C07282=1064.965,385.568,389.284,174.919,35.671,156.670
C07283=1064.957,385.321,389.325,174.915,35.664,156.668
C07284=1064.950,385.075,389.365,174.910,35.657,156.666
C07285=1064.943,384.828,389.405,174.904,35.650,156.665
C07286=1064.936,384.581,389.445,174.899,35.643,156.663
C07287=1064.928,384.334,389.485,174.895,35.636,156.662
C07288=1064.922,384.089,389.526,174.890,35.629,156.660
C07289=1064.914,383.842,389.566,174.884,35.621,156.658
C07290=1064.907,383.595,389.605,174.879,35.615,156.657
C07291=1064.900,383.348,389.646,174.875,35.608,156.655
C07292=1064.893,383.102,389.685,174.870,35.600,156.653
C07293=1064.886,382.855,389.726,174.865,35.594,156.652
C07294=1064.879,382.609,389.765,174.859,35.587,156.650
C07295=1064.871,382.362,389.805,174.855,35.580,156.649
C07296=1064.865,382.115,389.845,174.850,35.573,156.647
C07297=1064.857,381.868,389.885,174.845,35.566,156.645
C07298=1064.850,381.622,389.925,174.840,35.559,156.644
C07299=1064.843,381.376,389.965,174.835,35.552,156.642
C07300=1064.836,381.128,390.004,174.830,35.545,156.641
C07301=1064.829,380.882,390.044,174.825,35.538,156.639
C07302=1064.821,380.635,390.084,174.821,35.532,156.637
C07303=1064.814,380.389,390.123,174.816,35.525,156.636
C07304=1064.807,380.142,390.162,174.810,35.518,156.634
C07305=1064.799,379.895,390.202,174.805,35.511,156.633
C07306=1064.792,379.649,390.242,174.801,35.504,156.631
C07307=1064.785,379.401,390.281,174.796,35.498,156.630
C07308=1064.778,379.155,390.320,174.791,35.491,156.628
C07309=1064.771,378.908,390.359,174.787,35.484,156.627
C07310=1064.763,378.661,390.399,174.781,35.478,156.625
C07311=1064.756,378.415,390.439,174.776,35.471,156.624
C07312=1064.749,378.168,390.478,174.772,35.464,156.622
C07313=1064.742,377.921,390.517,174.767,35.458,156.621
C07314=1064.735,377.675,390.556,174.762,35.451,156.619
C07315=1064.728,377.428,390.595,174.758,35.444,156.617
C07316=1064.721,377.182,390.635,174.753,35.438,156.616
C07317=1064.713,376.934,390.674,174.748,35.432,156.615
C07318=1064.706,376.688,390.713,174.744,35.425,156.613
C07319=1064.700,376.441,390.752,174.738,35.418,156.611
C07320=1064.693,376.194,390.791,174.733,35.411,156.610
C07321=1064.685,375.947,390.831,174.729,35.405,156.609
C07322=1064.678,375.700,390.870,174.724,35.399,156.607
C07323=1064.671,375.454,390.909,174.719,35.392,156.605
C07324=1064.665,375.207,390.948,174.715,35.386,156.604
C07325=1064.657,374.961,390.987,174.710,35.379,156.603
C07326=1064.651,374.714,391.026,174.706,35.372,156.601
C07327=1064.644,374.467,391.065,174.701,35.366,156.600
C07328=1064.636,374.219,391.104,174.696,35.360,156.598
C07329=1064.630,373.973,391.142,174.692,35.353,156.597
C07330=1064.622,373.727,391.181,174.687,35.347,156.595
C07331=1064.616,373.481,391.220,174.683,35.341,156.594
C07332=1064.609,373.235,391.259,174.678,35.334,156.592
C07333=1064.602,372.988,391.298,174.673,35.328,156.591
C07334=1064.595,372.743,391.336,174.669,35.321,156.589
C07335=1064.588,372.496,391.375,174.664,35.315,156.588
C07336=1064.581,372.250,391.414,174.660,35.309,156.587
C07337=1064.574,372.002,391.452,174.655,35.302,156.585
C07338=1064.566,371.756,391.490,174.650,35.296,156.584
C07339=1064.560,371.509,391.529,174.646,35.290,156.582
C07340=1064.553,371.262,391.568,174.641,35.283,156.581
C07341=1064.545,371.016,391.606,174.637,35.277,156.579
C07342=1064.539,370.769,391.645,174.632,35.271,156.578
C07343=1064.532,370.521,391.683,174.627,35.265,156.577
C07344=1064.524,370.275,391.721,174.623,35.259,156.575
C07345=1064.518,370.028,391.760,174.618,35.253,156.574
C07346=1064.511,369.781,391.798,174.614,35.246,156.573
C07347=1064.504,369.534,391.837,174.609,35.240,156.571
C07348=1064.497,369.287,391.875,174.605,35.234,156.570
C07349=1064.490,369.040,391.913,174.600,35.228,156.568
C07350=1064.483,368.793,391.952,174.596,35.222,156.567
C07351=1064.476,368.546,391.990,174.591,35.215,156.566
C07352=1064.469,368.299,392.028,174.586,35.209,156.564
C07353=1064.462,368.052,392.066,174.582,35.204,156.563
C07354=1064.455,367.805,392.105,174.578,35.197,156.562
C07355=1064.449,367.559,392.142,174.574,35.191,156.560
C07356=1064.442,367.312,392.181,174.569,35.185,156.559
C07357=1064.435,367.065,392.219,174.565,35.179,156.557
C07358=1064.428,366.818,392.258,174.560,35.173,156.556
C07359=1064.421,366.571,392.295,174.556,35.167,156.555
C07360=1064.414,366.323,392.333,174.551,35.161,156.553
C07361=1064.407,366.077,392.371,174.547,35.155,156.552
C07362=1064.401,365.830,392.409,174.542,35.149,156.551
C07363=1064.393,365.583,392.447,174.539,35.143,156.549
C07364=1064.387,365.336,392.486,174.534,35.137,156.548
C07365=1064.380,365.089,392.524,174.530,35.131,156.547
C07366=1064.373,364.842,392.561,174.525,35.125,156.545
C07367=1064.367,364.595,392.599,174.521,35.119,156.544
C07368=1064.359,364.348,392.637,174.516,35.113,156.543
C07369=1064.353,364.101,392.675,174.512,35.107,156.541
C07370=1064.346,363.854,392.713,174.508,35.101,156.540
C07371=1064.339,363.607,392.750,174.504,35.095,156.539
C07372=1064.332,363.360,392.788,174.499,35.089,156.537
C07373=1064.325,363.113,392.826,174.495,35.084,156.536
C07374=1064.318,362.866,392.863,174.490,35.078,156.535
C07375=1064.311,362.619,392.900,174.486,35.072,156.533
C07376=1064.305,362.372,392.938,174.482,35.066,156.532
C07377=1064.298,362.125,392.976,174.478,35.060,156.531
C07378=1064.290,361.877,393.013,174.473,35.055,156.530
C07379=1064.284,361.631,393.051,174.469,35.048,156.528
C07380=1064.277,361.384,393.089,174.464,35.043,156.527
C07381=1064.270,361.136,393.126,174.461,35.037,156.526
C07382=1064.264,360.889,393.163,174.456,35.031,156.525
C07383=1064.256,360.642,393.200,174.452,35.026,156.523
C07384=1064.250,360.395,393.238,174.447,35.020,156.522
C07385=1064.243,360.158,393.274,174.444,35.014,156.521
C07386=1064.237,359.920,393.310,174.439,35.009,156.520
C07387=1064.230,359.683,393.346,174.435,35.004,156.518
C07388=1064.224,359.445,393.382,174.431,34.998,156.517
C07389=1064.217,359.208,393.417,174.427,34.992,156.516
C07390=1064.211,358.970,393.453,174.424,34.987,156.515
C07391=1064.204,358.733,393.489,174.419,34.981,156.514
C07392=1064.195,358.386,393.541,174.414,34.974,156.512
C07393=1064.185,358.030,393.595,174.407,34.966,156.510
C07394=1064.178,357.782,393.632,174.403,34.960,156.509
C07395=1064.171,357.535,393.669,174.399,34.954,156.508
C07396=1064.165,357.288,393.706,174.395,34.948,156.506
C07397=1064.157,357.041,393.743,174.390,34.943,156.505
C07398=1064.151,356.793,393.780,174.387,34.938,156.504
C07399=1064.144,356.546,393.817,174.382,34.932,156.503
C07400=1064.137,356.299,393.854,174.378,34.926,156.502
C07401=1064.130,356.052,393.891,174.373,34.921,156.500
C07402=1064.124,355.805,393.928,174.370,34.915,156.499
C07403=1064.117,355.557,393.965,174.366,34.910,156.498
C07404=1064.111,355.310,394.001,174.361,34.904,156.497
C07405=1064.103,355.063,394.039,174.358,34.899,156.496
C07406=1064.097,354.816,394.075,174.353,34.893,156.494
C07407=1064.090,354.568,394.112,174.349,34.887,156.493
C07408=1064.083,354.322,394.149,174.346,34.882,156.492
C07409=1064.076,354.074,394.186,174.341,34.877,156.491
C07410=1064.070,353.827,394.222,174.337,34.871,156.489
C07411=1064.064,353.580,394.259,174.333,34.866,156.488
C07412=1064.056,353.333,394.296,174.329,34.860,156.487
C07413=1064.050,353.086,394.333,174.324,34.855,156.486
C07414=1064.043,352.838,394.369,174.321,34.849,156.485
C07415=1064.037,352.591,394.406,174.317,34.844,156.484
C07416=1064.031,352.344,394.442,174.312,34.838,156.482
C07417=1064.024,352.096,394.479,174.309,34.833,156.481
C07418=1064.017,351.849,394.516,174.304,34.828,156.480
C07419=1064.010,351.602,394.551,174.301,34.822,156.479
C07420=1064.003,351.355,394.588,174.297,34.817,156.478
C07421=1063.997,351.108,394.625,174.292,34.811,156.477
C07422=1063.990,350.860,394.661,174.289,34.806,156.475
C07423=1063.983,350.613,394.697,174.285,34.801,156.474
C07424=1063.977,350.366,394.734,174.280,34.795,156.473
C07425=1063.970,350.118,394.771,174.277,34.790,156.472
C07426=1063.963,349.871,394.807,174.272,34.785,156.471
C07427=1063.956,349.625,394.843,174.269,34.779,156.470
C07428=1063.950,349.377,394.879,174.265,34.774,156.468
C07429=1063.943,349.129,394.915,174.260,34.769,156.467
C07430=1063.936,348.882,394.951,174.257,34.764,156.466
C07431=1063.930,348.635,394.988,174.253,34.759,156.465
C07432=1063.923,348.388,395.025,174.249,34.753,156.464
C07433=1063.917,348.140,395.060,174.245,34.748,156.463
C07434=1063.910,347.893,395.096,174.241,34.743,156.462
C07435=1063.903,347.646,395.133,174.237,34.738,156.461
C07436=1063.897,347.398,395.169,174.233,34.732,156.459
C07437=1063.890,347.151,395.205,174.229,34.727,156.458
C07438=1063.883,346.904,395.241,174.225,34.722,156.457
C07439=1063.877,346.656,395.276,174.222,34.717,156.456
C07440=1063.870,346.409,395.313,174.217,34.712,156.455
C07441=1063.859,345.994,395.373,174.211,34.702,156.453
C07442=1063.848,345.577,395.433,174.204,34.694,156.451
C07443=1063.837,345.161,395.494,174.198,34.685,156.449
C07444=1063.826,344.745,395.554,174.192,34.677,156.448
C07445=1063.819,344.498,395.590,174.188,34.671,156.446
C07446=1063.813,344.250,395.626,174.183,34.666,156.445
C07447=1063.806,344.004,395.662,174.180,34.661,156.444
C07448=1063.800,343.756,395.698,174.176,34.656,156.443
C07449=1063.793,343.508,395.733,174.172,34.651,156.442
C07450=1063.787,343.261,395.769,174.168,34.646,156.441
C07451=1063.780,343.013,395.805,174.165,34.641,156.440
C07452=1063.773,342.766,395.840,174.160,34.636,156.439
C07453=1063.767,342.518,395.876,174.157,34.631,156.438
C07454=1063.760,342.272,395.911,174.154,34.626,156.437
C07455=1063.753,342.024,395.947,174.149,34.621,156.436
C07456=1063.747,341.777,395.982,174.146,34.615,156.434
C07457=1063.740,341.529,396.017,174.142,34.611,156.434
C07458=1063.733,341.282,396.053,174.138,34.606,156.432
C07459=1063.727,341.035,396.089,174.134,34.600,156.431
C07460=1063.720,340.787,396.124,174.131,34.596,156.430
C07461=1063.714,340.540,396.160,174.126,34.591,156.429
C07462=1063.707,340.292,396.195,174.123,34.585,156.428
C07463=1063.701,340.045,396.230,174.119,34.581,156.427
C07464=1063.694,339.798,396.265,174.115,34.575,156.426
C07465=1063.688,339.550,396.301,174.111,34.571,156.425
C07466=1063.681,339.303,396.336,174.108,34.566,156.424
C07467=1063.674,339.055,396.371,174.105,34.560,156.423
C07468=1063.668,338.808,396.407,174.100,34.556,156.422
C07469=1063.662,338.560,396.442,174.097,34.551,156.421
C07470=1063.655,338.313,396.477,174.093,34.546,156.420
C07471=1063.649,338.065,396.513,174.089,34.541,156.419
C07472=1063.642,337.818,396.548,174.086,34.536,156.418
C07473=1063.635,337.570,396.583,174.082,34.531,156.417
C07474=1063.628,337.323,396.618,174.078,34.526,156.416
C07475=1063.622,337.075,396.654,174.074,34.521,156.415
C07476=1063.617,336.828,396.688,174.071,34.516,156.414
C07477=1063.610,336.581,396.723,174.068,34.512,156.413
C07478=1063.603,336.333,396.758,174.063,34.506,156.411
C07479=1063.596,336.086,396.794,174.060,34.502,156.410
C07480=1063.590,335.838,396.828,174.056,34.497,156.409
C07481=1063.583,335.591,396.863,174.052,34.492,156.408
C07482=1063.576,335.343,396.898,174.049,34.487,156.407
C07483=1063.570,335.096,396.933,174.045,34.483,156.406
C07484=1063.563,334.848,396.968,174.042,34.477,156.405
C07485=1063.558,334.601,397.003,174.038,34.473,156.404
C07486=1063.551,334.354,397.038,174.034,34.468,156.403
C07487=1063.544,334.106,397.073,174.031,34.463,156.402
C07488=1063.538,333.858,397.108,174.026,34.458,156.401
C07489=1063.531,333.610,397.142,174.023,34.454,156.400
C07490=1063.525,333.364,397.177,174.020,34.449,156.399
C07491=1063.519,333.116,397.211,174.016,34.444,156.398
C07492=1063.512,332.868,397.247,174.012,34.439,156.397
C07493=1063.505,332.631,397.280,174.009,34.434,156.396
C07494=1063.499,332.393,397.313,174.006,34.430,156.395
C07495=1063.493,332.155,397.347,174.003,34.426,156.395
C07496=1063.487,331.917,397.380,173.998,34.421,156.394
C07497=1063.480,331.680,397.413,173.995,34.416,156.393
C07498=1063.475,331.441,397.446,173.992,34.412,156.392
C07499=1063.468,331.204,397.480,173.989,34.407,156.391
C07500=1063.462,330.966,397.513,173.985,34.402,156.390
C07501=1063.456,330.718,397.547,173.981,34.398,156.389
C07502=1063.449,330.471,397.582,173.978,34.393,156.388
C07503=1063.442,330.223,397.616,173.975,34.388,156.387
C07504=1063.436,329.976,397.650,173.970,34.384,156.386
C07505=1063.429,329.728,397.684,173.967,34.379,156.385
C07506=1063.423,329.481,397.719,173.964,34.375,156.384
C07507=1063.415,329.233,397.753,173.960,34.370,156.383
C07508=1063.410,328.986,397.787,173.956,34.366,156.382
C07509=1063.403,328.738,397.822,173.953,34.361,156.381
C07510=1063.396,328.490,397.856,173.950,34.356,156.380
C07511=1063.389,328.243,397.891,173.946,34.351,156.379
C07512=1063.383,327.995,397.925,173.942,34.347,156.378
C07513=1063.376,327.748,397.959,173.939,34.342,156.377
C07514=1063.370,327.500,397.993,173.935,34.338,156.376
C07515=1063.364,327.252,398.027,173.932,34.333,156.375
C07516=1063.357,327.005,398.061,173.928,34.329,156.374
C07517=1063.350,326.757,398.095,173.925,34.324,156.373
C07518=1063.343,326.510,398.129,173.921,34.319,156.372
C07519=1063.337,326.262,398.163,173.918,34.315,156.371
C07520=1063.331,326.014,398.197,173.914,34.311,156.371
C07521=1063.324,325.767,398.231,173.911,34.306,156.370
C07522=1063.317,325.519,398.266,173.907,34.301,156.369
C07523=1063.311,325.272,398.299,173.904,34.296,156.368
C07524=1063.304,325.024,398.333,173.901,34.292,156.367
C07525=1063.299,324.777,398.367,173.897,34.288,156.366
C07526=1063.291,324.529,398.401,173.893,34.283,156.365
C07527=1063.285,324.281,398.436,173.890,34.278,156.364
C07528=1063.279,324.033,398.468,173.887,34.274,156.363
C07529=1063.272,323.785,398.503,173.883,34.269,156.362
C07530=1063.266,323.538,398.537,173.880,34.265,156.361
C07531=1063.259,323.290,398.571,173.876,34.260,156.360
C07532=1063.253,323.043,398.605,173.873,34.256,156.359
C07533=1063.246,322.795,398.639,173.870,34.251,156.358
C07534=1063.240,322.547,398.672,173.866,34.247,156.357
C07535=1063.233,322.300,398.706,173.863,34.242,156.357
C07536=1063.227,322.053,398.740,173.859,34.238,156.356
C07537=1063.221,321.806,398.773,173.856,34.233,156.355
C07538=1063.215,321.557,398.807,173.852,34.229,156.354
C07539=1063.209,321.310,398.841,173.849,34.224,156.353
C07540=1063.202,321.062,398.875,173.846,34.220,156.352
C07541=1063.196,320.814,398.908,173.843,34.215,156.351
C07542=1063.189,320.566,398.942,173.839,34.211,156.350
C07543=1063.183,320.319,398.975,173.835,34.206,156.349
C07544=1063.177,320.072,399.009,173.832,34.202,156.348
C07545=1063.170,319.824,399.043,173.829,34.197,156.347
C07546=1063.164,319.576,399.076,173.826,34.193,156.346
C07547=1063.157,319.328,399.110,173.823,34.188,156.346
C07548=1063.151,319.080,399.143,173.819,34.184,156.345
C07549=1063.145,318.839,399.176,173.815,34.179,156.344
C07550=1063.139,318.599,399.209,173.812,34.175,156.343
C07551=1063.133,318.358,399.242,173.809,34.171,156.342
C07552=1063.127,318.118,399.274,173.806,34.167,156.341
C07553=1063.121,317.878,399.306,173.802,34.162,156.340
C07554=1063.115,317.637,399.338,173.799,34.158,156.339
C07555=1063.109,317.396,399.371,173.796,34.154,156.338
C07556=1063.103,317.155,399.404,173.793,34.149,156.338
C07557=1063.096,316.908,399.437,173.790,34.145,156.337
C07558=1063.091,316.660,399.470,173.786,34.140,156.336
C07559=1063.084,316.412,399.503,173.783,34.135,156.335
C07560=1063.078,316.164,399.538,173.780,34.131,156.334
C07561=1063.071,315.917,399.570,173.777,34.127,156.333
C07562=1063.066,315.669,399.604,173.774,34.122,156.332
C07563=1063.059,315.421,399.637,173.770,34.118,156.331
C07564=1063.052,315.174,399.670,173.767,34.114,156.330
C07565=1063.047,314.926,399.703,173.763,34.109,156.329
C07566=1063.040,314.679,399.737,173.760,34.105,156.329
C07567=1063.035,314.431,399.770,173.757,34.100,156.328
C07568=1063.028,314.183,399.803,173.753,34.096,156.327
C07569=1063.022,313.935,399.837,173.750,34.091,156.326
C07570=1063.016,313.687,399.869,173.747,34.087,156.325
C07571=1063.010,313.440,399.902,173.744,34.083,156.324
C07572=1063.002,313.192,399.936,173.741,34.079,156.323
C07573=1062.996,312.944,399.969,173.738,34.074,156.322
C07574=1062.990,312.697,400.002,173.734,34.070,156.321
C07575=1062.983,312.449,400.034,173.731,34.066,156.321
C07576=1062.976,312.201,400.067,173.728,34.062,156.320
C07577=1062.970,311.953,400.100,173.725,34.057,156.319
C07578=1062.963,311.706,400.132,173.721,34.053,156.318
C07579=1062.957,311.458,400.165,173.718,34.048,156.317
C07580=1062.951,311.211,400.198,173.714,34.044,156.316
C07581=1062.944,310.962,400.231,173.711,34.040,156.315
C07582=1062.938,310.715,400.264,173.708,34.036,156.315
C07583=1062.932,310.467,400.296,173.705,34.032,156.314
C07584=1062.925,310.219,400.328,173.702,34.027,156.313
C07585=1062.919,309.971,400.361,173.699,34.023,156.312
C07586=1062.912,309.723,400.394,173.695,34.019,156.311
C07587=1062.905,309.476,400.426,173.692,34.015,156.310
C07588=1062.899,309.228,400.459,173.689,34.010,156.310
C07589=1062.893,308.981,400.492,173.686,34.006,156.309
C07590=1062.887,308.732,400.524,173.683,34.002,156.308
C07591=1062.880,308.485,400.557,173.680,33.998,156.307
C07592=1062.874,308.237,400.589,173.676,33.993,156.306
C07593=1062.868,307.990,400.622,173.673,33.989,156.305
C07594=1062.861,307.742,400.655,173.670,33.985,156.304
C07595=1062.855,307.494,400.686,173.667,33.981,156.304
C07596=1062.848,307.247,400.719,173.664,33.977,156.303
C07597=1062.842,306.999,400.752,173.661,33.972,156.302
C07598=1062.835,306.750,400.784,173.657,33.968,156.301
C07599=1062.829,306.502,400.817,173.654,33.964,156.300
C07600=1062.823,306.255,400.850,173.651,33.960,156.299
C07601=1062.816,306.007,400.881,173.648,33.955,156.298
C07602=1062.810,305.759,400.914,173.645,33.951,156.298
C07603=1062.804,305.512,400.947,173.642,33.947,156.297
C07604=1062.798,305.264,400.978,173.638,33.943,156.296
C07605=1062.791,305.025,401.010,173.635,33.939,156.295
C07606=1062.785,304.786,401.041,173.632,33.935,156.294
C07607=1062.779,304.547,401.072,173.629,33.931,156.294
C07608=1062.774,304.308,401.103,173.626,33.927,156.293
C07609=1062.767,304.070,401.135,173.623,33.922,156.292
C07610=1062.761,303.831,401.166,173.620,33.918,156.291
C07611=1062.755,303.592,401.196,173.618,33.915,156.290
C07612=1062.750,303.354,401.227,173.614,33.911,156.290
C07613=1062.743,303.106,401.259,173.611,33.906,156.289
C07614=1062.737,302.858,401.291,173.608,33.902,156.288
C07615=1062.731,302.611,401.324,173.605,33.898,156.287
C07616=1062.725,302.362,401.356,173.602,33.894,156.286
C07617=1062.719,302.115,401.389,173.599,33.889,156.285
C07618=1062.712,301.867,401.420,173.595,33.885,156.284
C07619=1062.706,301.619,401.452,173.592,33.881,156.284
C07620=1062.700,301.372,401.485,173.589,33.877,156.283
C07621=1062.694,301.123,401.517,173.586,33.872,156.282
C07622=1062.688,300.876,401.548,173.583,33.868,156.281
C07623=1062.681,300.628,401.581,173.581,33.864,156.280
C07624=1062.675,300.380,401.613,173.578,33.860,156.279
C07625=1062.669,300.132,401.645,173.575,33.856,156.279
C07626=1062.663,299.885,401.677,173.571,33.852,156.278
C07627=1062.657,299.637,401.709,173.568,33.847,156.277
C07628=1062.651,299.389,401.741,173.565,33.843,156.276
C07629=1062.645,299.140,401.773,173.562,33.839,156.275
C07630=1062.638,298.892,401.804,173.559,33.835,156.274
C07631=1062.632,298.646,401.837,173.556,33.831,156.274
C07632=1062.626,298.397,401.869,173.553,33.826,156.273
C07633=1062.620,298.149,401.901,173.550,33.822,156.272
C07634=1062.614,297.902,401.932,173.547,33.818,156.271
C07635=1062.608,297.654,401.964,173.544,33.814,156.270
C07636=1062.602,297.405,401.996,173.541,33.810,156.270
C07637=1062.595,297.158,402.028,173.538,33.806,156.269
C07638=1062.590,296.911,402.060,173.535,33.801,156.268
C07639=1062.583,296.663,402.091,173.532,33.797,156.267
C07640=1062.577,296.415,402.123,173.530,33.793,156.266
C07641=1062.571,296.167,402.155,173.526,33.790,156.265
C07642=1062.565,295.918,402.187,173.523,33.785,156.265
C07643=1062.558,295.671,402.218,173.520,33.781,156.264
C07644=1062.552,295.423,402.250,173.517,33.777,156.263
C07645=1062.546,295.175,402.281,173.514,33.773,156.262
C07646=1062.541,294.927,402.312,173.511,33.769,156.261
C07647=1062.534,294.679,402.344,173.508,33.765,156.261
C07648=1062.527,294.431,402.375,173.506,33.761,156.260
C07649=1062.521,294.183,402.407,173.502,33.757,156.259
C07650=1062.515,293.936,402.438,173.499,33.752,156.258
C07651=1062.508,293.688,402.470,173.496,33.749,156.257
C07652=1062.502,293.440,402.502,173.493,33.745,156.257
C07653=1062.496,293.191,402.532,173.490,33.740,156.256
C07654=1062.490,292.944,402.563,173.488,33.736,156.255
C07655=1062.484,292.696,402.595,173.485,33.733,156.254
C07656=1062.477,292.448,402.627,173.482,33.728,156.253
C07657=1062.471,292.201,402.658,173.479,33.724,156.253
C07658=1062.465,291.952,402.689,173.475,33.720,156.252
C07659=1062.459,291.704,402.721,173.472,33.716,156.251
C07660=1062.452,291.457,402.752,173.470,33.712,156.250
C07661=1062.447,291.225,402.780,173.467,33.709,156.250
C07662=1062.440,290.994,402.810,173.464,33.704,156.249
C07663=1062.435,290.763,402.838,173.462,33.701,156.248
C07664=1062.429,290.532,402.868,173.459,33.697,156.247
C07665=1062.423,290.300,402.897,173.456,33.694,156.247
C07666=1062.417,290.069,402.926,173.454,33.689,156.246
C07667=1062.412,289.838,402.955,173.450,33.686,156.245
C07668=1062.406,289.607,402.984,173.448,33.682,156.244
C07669=1062.400,289.359,403.015,173.445,33.678,156.244
C07670=1062.394,289.111,403.047,173.442,33.674,156.243
C07671=1062.388,288.862,403.077,173.439,33.670,156.242
C07672=1062.381,288.615,403.109,173.437,33.666,156.241
C07673=1062.375,288.366,403.139,173.434,33.662,156.240
C07674=1062.369,288.119,403.170,173.431,33.658,156.240
C07675=1062.362,287.871,403.201,173.428,33.654,156.239
C07676=1062.356,287.623,403.232,173.425,33.650,156.238
C07677=1062.350,287.375,403.263,173.422,33.646,156.237
C07678=1062.343,287.127,403.294,173.419,33.642,156.237
C07679=1062.337,286.879,403.325,173.416,33.638,156.236
C07680=1062.331,286.631,403.355,173.413,33.634,156.235
C07681=1062.324,286.383,403.387,173.411,33.630,156.234
C07682=1062.318,286.135,403.417,173.408,33.626,156.233
C07683=1062.312,285.887,403.449,173.405,33.622,156.233
C07684=1062.306,285.639,403.479,173.402,33.618,156.232
C07685=1062.300,285.390,403.510,173.399,33.614,156.231
C07686=1062.294,285.143,403.541,173.397,33.610,156.230
C07687=1062.288,284.895,403.572,173.394,33.606,156.230
C07688=1062.282,284.647,403.602,173.390,33.602,156.229
C07689=1062.275,284.398,403.633,173.388,33.599,156.228
C07690=1062.269,284.152,403.663,173.385,33.594,156.227
C07691=1062.262,283.903,403.694,173.382,33.590,156.226
C07692=1062.256,283.655,403.725,173.379,33.586,156.226
C07693=1062.250,283.407,403.755,173.377,33.582,156.225
C07694=1062.244,283.159,403.786,173.374,33.579,156.224
C07695=1062.237,282.911,403.817,173.371,33.574,156.223
C07696=1062.232,282.663,403.847,173.368,33.570,156.223
C07697=1062.225,282.415,403.878,173.366,33.567,156.222
C07698=1062.219,282.167,403.908,173.363,33.562,156.221
C07699=1062.213,281.919,403.939,173.359,33.559,156.220
C07700=1062.207,281.670,403.970,173.357,33.555,156.220
C07701=1062.201,281.423,404.000,173.354,33.550,156.219
C07702=1062.195,281.175,404.031,173.351,33.547,156.218
C07703=1062.189,280.927,404.062,173.349,33.543,156.217
C07704=1062.183,280.679,404.092,173.346,33.539,156.217
C07705=1062.176,280.431,404.123,173.343,33.535,156.216
C07706=1062.171,280.183,404.153,173.340,33.530,156.215
C07707=1062.164,279.934,404.184,173.338,33.527,156.214
C07708=1062.158,279.687,404.214,173.335,33.523,156.213
C07709=1062.152,279.439,404.244,173.332,33.519,156.213
C07710=1062.145,279.190,404.275,173.330,33.515,156.212
C07711=1062.140,278.942,404.304,173.326,33.511,156.211
C07712=1062.133,278.694,404.334,173.323,33.507,156.210
C07713=1062.127,278.446,404.365,173.321,33.503,156.210
C07714=1062.121,278.198,404.395,173.318,33.499,156.209
C07715=1062.115,277.950,404.426,173.315,33.495,156.208
C07716=1062.108,277.702,404.456,173.313,33.491,156.207
C07717=1062.103,277.476,404.484,173.310,33.488,156.207
C07718=1062.097,277.250,404.511,173.308,33.485,156.206
C07719=1062.091,277.024,404.538,173.305,33.481,156.205
C07720=1062.085,276.799,404.566,173.303,33.477,156.205
C07721=1062.081,276.572,404.593,173.301,33.474,156.204
C07722=1062.075,276.347,404.620,173.298,33.470,156.203
C07723=1062.070,276.121,404.648,173.296,33.466,156.203
C07724=1062.063,275.895,404.675,173.293,33.463,156.202
C07725=1062.057,275.647,404.706,173.291,33.459,156.201
C07726=1062.052,275.398,404.735,173.287,33.455,156.200
C07727=1062.045,275.150,404.765,173.284,33.451,156.200
C07728=1062.039,274.902,404.796,173.282,33.447,156.199
C07729=1062.033,274.655,404.826,173.279,33.443,156.198
C07730=1062.027,274.406,404.855,173.276,33.439,156.197
C07731=1062.020,274.158,404.886,173.274,33.436,156.197
C07732=1062.014,273.910,404.915,173.271,33.431,156.196
C07733=1062.008,273.662,404.945,173.269,33.428,156.195
C07734=1062.002,273.413,404.976,173.266,33.424,156.194
C07735=1061.995,273.165,405.005,173.263,33.420,156.194
C07736=1061.990,272.917,405.035,173.261,33.416,156.193
C07737=1061.983,272.669,405.064,173.258,33.412,156.192
C07738=1061.977,272.421,405.095,173.256,33.408,156.191
C07739=1061.970,272.173,405.125,173.253,33.404,156.191
C07740=1061.965,271.925,405.155,173.250,33.400,156.190
C07741=1061.958,271.677,405.184,173.247,33.396,156.189
C07742=1061.952,271.428,405.214,173.244,33.393,156.188
C07743=1061.946,271.180,405.243,173.242,33.388,156.188
C07744=1061.940,270.932,405.274,173.239,33.385,156.187
C07745=1061.934,270.684,405.303,173.236,33.381,156.186
C07746=1061.928,270.436,405.333,173.234,33.377,156.185
C07747=1061.921,270.187,405.362,173.231,33.373,156.185
C07748=1061.915,269.940,405.393,173.229,33.369,156.184
C07749=1061.909,269.691,405.422,173.226,33.365,156.183
C07750=1061.904,269.443,405.451,173.223,33.361,156.182
C07751=1061.897,269.196,405.481,173.221,33.357,156.182
C07752=1061.891,268.947,405.510,173.218,33.354,156.181
C07753=1061.885,268.698,405.540,173.216,33.350,156.180
C07754=1061.878,268.451,405.570,173.213,33.346,156.179
C07755=1061.873,268.202,405.600,173.211,33.342,156.179
C07756=1061.866,267.954,405.629,173.208,33.338,156.178
C07757=1061.860,267.707,405.658,173.205,33.334,156.177
C07758=1061.854,267.458,405.688,173.203,33.330,156.176
C07759=1061.848,267.209,405.718,173.199,33.327,156.176
C07760=1061.841,266.961,405.747,173.197,33.323,156.175
C07761=1061.835,266.714,405.776,173.194,33.319,156.174
C07762=1061.829,266.465,405.806,173.192,33.315,156.173
C07763=1061.823,266.217,405.835,173.189,33.311,156.173
C07764=1061.817,265.969,405.864,173.187,33.307,156.172
C07765=1061.811,265.721,405.894,173.184,33.303,156.171
C07766=1061.805,265.472,405.923,173.181,33.299,156.170
C07767=1061.798,265.224,405.953,173.179,33.296,156.170
C07768=1061.792,264.976,405.982,173.176,33.291,156.169
C07769=1061.786,264.728,406.012,173.174,33.288,156.168
C07770=1061.780,264.480,406.041,173.171,33.284,156.168
C07771=1061.774,264.231,406.070,173.169,33.280,156.167
C07772=1061.768,263.983,406.099,173.166,33.276,156.166
C07773=1061.763,263.759,406.125,173.164,33.273,156.165
C07774=1061.756,263.535,406.152,173.162,33.269,156.165
C07775=1061.752,263.311,406.178,173.159,33.265,156.164
C07776=1061.746,263.087,406.205,173.157,33.262,156.163
C07777=1061.740,262.863,406.231,173.155,33.259,156.163
C07778=1061.734,262.639,406.257,173.153,33.256,156.162
C07779=1061.728,262.415,406.283,173.150,33.252,156.161
C07780=1061.722,262.191,406.309,173.148,33.248,156.161
C07781=1061.716,261.943,406.338,173.146,33.245,156.160
C07782=1061.710,261.694,406.367,173.143,33.241,156.159
C07783=1061.704,261.446,406.396,173.139,33.237,156.159
C07784=1061.698,261.198,406.425,173.137,33.233,156.158
C07785=1061.691,260.950,406.454,173.134,33.229,156.157
C07786=1061.685,260.702,406.483,173.132,33.226,156.156
C07787=1061.679,260.453,406.512,173.129,33.222,156.156
C07788=1061.673,260.205,406.541,173.127,33.218,156.155
C07789=1061.667,259.957,406.569,173.124,33.214,156.154
C07790=1061.660,259.708,406.598,173.122,33.210,156.154
C07791=1061.653,259.461,406.627,173.119,33.207,156.153
C07792=1061.647,259.212,406.656,173.117,33.203,156.152
C07793=1061.641,258.964,406.685,173.114,33.199,156.151
C07794=1061.635,258.716,406.713,173.112,33.195,156.151
C07795=1061.629,258.467,406.742,173.110,33.191,156.150
C07796=1061.622,258.219,406.771,173.107,33.187,156.149
C07797=1061.617,257.971,406.800,173.105,33.184,156.149
C07798=1061.610,257.722,406.829,173.102,33.180,156.148
C07799=1061.604,257.474,406.858,173.100,33.176,156.147
C07800=1061.598,257.226,406.886,173.097,33.172,156.146
C07801=1061.592,256.977,406.915,173.095,33.168,156.146
C07802=1061.585,256.730,406.944,173.092,33.164,156.145
C07803=1061.579,256.481,406.972,173.090,33.161,156.144
C07804=1061.573,256.233,407.001,173.087,33.157,156.143
C07805=1061.566,255.985,407.030,173.085,33.153,156.143
C07806=1061.560,255.736,407.058,173.082,33.149,156.142
C07807=1061.554,255.488,407.087,173.080,33.145,156.141
C07808=1061.549,255.240,407.115,173.078,33.141,156.140
C07809=1061.543,254.991,407.144,173.075,33.137,156.140
C07810=1061.536,254.743,407.172,173.073,33.134,156.139
C07811=1061.530,254.495,407.201,173.070,33.130,156.138
C07812=1061.523,254.247,407.230,173.068,33.126,156.138
C07813=1061.517,253.998,407.258,173.065,33.122,156.137
C07814=1061.511,253.750,407.287,173.063,33.118,156.136
C07815=1061.505,253.501,407.316,173.061,33.114,156.135
C07816=1061.500,253.253,407.344,173.058,33.111,156.135
C07817=1061.493,253.005,407.372,173.056,33.106,156.134
C07818=1061.487,252.757,407.401,173.053,33.103,156.133
C07819=1061.481,252.508,407.430,173.050,33.099,156.133
C07820=1061.475,252.260,407.458,173.048,33.095,156.132
C07821=1061.469,252.012,407.487,173.045,33.091,156.131
C07822=1061.463,251.763,407.515,173.043,33.087,156.130
C07823=1061.457,251.515,407.543,173.040,33.083,156.130
C07824=1061.450,251.267,407.572,173.038,33.079,156.129
C07825=1061.444,251.018,407.600,173.036,33.076,156.128
C07826=1061.438,250.769,407.628,173.033,33.072,156.127
C07827=1061.433,250.522,407.657,173.031,33.068,156.127
C07828=1061.426,250.274,407.685,173.028,33.064,156.126
C07829=1061.421,250.048,407.711,173.026,33.061,156.125
C07830=1061.415,249.823,407.737,173.024,33.057,156.125
C07831=1061.409,249.598,407.762,173.022,33.053,156.124
C07832=1061.405,249.372,407.788,173.020,33.050,156.123
C07833=1061.399,249.148,407.813,173.018,33.046,156.123
C07834=1061.394,248.923,407.839,173.016,33.043,156.122
C07835=1061.389,248.698,407.865,173.013,33.039,156.121
C07836=1061.383,248.473,407.891,173.011,33.036,156.121
C07837=1061.377,248.224,407.919,173.009,33.031,156.120
C07838=1061.371,247.977,407.946,173.007,33.028,156.119
C07839=1061.365,247.728,407.975,173.004,33.024,156.118
C07840=1061.359,247.479,408.003,173.002,33.020,156.118
C07841=1061.353,247.231,408.031,172.999,33.016,156.117
C07842=1061.346,246.983,408.060,172.997,33.012,156.116
C07843=1061.341,246.734,408.088,172.995,33.008,156.115
C07844=1061.335,246.486,408.116,172.992,33.004,156.115
C07845=1061.329,246.238,408.144,172.990,33.000,156.114
C07846=1061.323,245.989,408.172,172.988,32.997,156.113
C07847=1061.317,245.740,408.200,172.985,32.992,156.112
C07848=1061.311,245.493,408.228,172.983,32.989,156.112
C07849=1061.305,245.244,408.256,172.981,32.985,156.111
C07850=1061.298,244.996,408.284,172.978,32.981,156.110
C07851=1061.293,244.747,408.312,172.976,32.977,156.110
C07852=1061.286,244.499,408.339,172.974,32.973,156.109
C07853=1061.280,244.250,408.368,172.971,32.969,156.108
C07854=1061.275,244.002,408.396,172.969,32.965,156.107
C07855=1061.268,243.754,408.423,172.967,32.962,156.107
C07856=1061.262,243.505,408.452,172.964,32.957,156.106
C07857=1061.256,243.257,408.479,172.962,32.954,156.105
C07858=1061.250,243.009,408.507,172.960,32.950,156.104
C07859=1061.243,242.760,408.535,172.958,32.946,156.104
C07860=1061.238,242.512,408.563,172.955,32.942,156.103
C07861=1061.231,242.264,408.591,172.953,32.938,156.102
C07862=1061.226,242.016,408.619,172.951,32.934,156.102
C07863=1061.220,241.767,408.646,172.948,32.931,156.101
C07864=1061.213,241.518,408.673,172.946,32.926,156.100
C07865=1061.207,241.269,408.702,172.944,32.923,156.099
C07866=1061.201,241.022,408.729,172.941,32.919,156.099
C07867=1061.194,240.773,408.757,172.939,32.915,156.098
C07868=1061.189,240.524,408.784,172.937,32.911,156.097
C07869=1061.182,240.276,408.812,172.934,32.907,156.096
C07870=1061.176,240.028,408.840,172.932,32.904,156.096
C07871=1061.170,239.780,408.867,172.930,32.899,156.095
C07872=1061.164,239.530,408.895,172.928,32.896,156.094
C07873=1061.158,239.283,408.922,172.925,32.892,156.094
C07874=1061.151,239.034,408.950,172.923,32.888,156.093
C07875=1061.146,238.785,408.977,172.921,32.884,156.092
C07876=1061.140,238.537,409.005,172.918,32.880,156.091
C07877=1061.133,238.289,409.032,172.916,32.876,156.091
C07878=1061.127,238.040,409.059,172.914,32.873,156.090
C07879=1061.121,237.792,409.087,172.912,32.869,156.089
C07880=1061.115,237.544,409.115,172.909,32.865,156.088
C07881=1061.109,237.295,409.142,172.907,32.861,156.088
C07882=1061.102,237.046,409.169,172.905,32.857,156.087
C07883=1061.096,236.799,409.197,172.903,32.853,156.086
C07884=1061.090,236.549,409.224,172.900,32.849,156.086
C07885=1061.084,236.322,409.249,172.898,32.846,156.085
C07886=1061.079,236.093,409.274,172.896,32.842,156.084
C07887=1061.073,235.865,409.300,172.894,32.839,156.084
C07888=1061.068,235.637,409.324,172.892,32.835,156.083
C07889=1061.063,235.409,409.350,172.890,32.832,156.082
C07890=1061.057,235.181,409.375,172.888,32.828,156.082
C07891=1061.052,234.953,409.400,172.886,32.824,156.081
C07892=1061.045,234.725,409.425,172.884,32.821,156.080
C07893=1061.040,234.476,409.453,172.882,32.817,156.080
C07894=1061.034,234.227,409.479,172.879,32.813,156.079
C07895=1061.027,233.979,409.507,172.877,32.809,156.078
C07896=1061.021,233.731,409.534,172.875,32.805,156.077
C07897=1061.015,233.482,409.562,172.873,32.801,156.077
C07898=1061.009,233.234,409.588,172.871,32.797,156.076
C07899=1061.004,232.985,409.615,172.869,32.794,156.075
C07900=1060.997,232.737,409.643,172.867,32.789,156.074
C07901=1060.991,232.488,409.670,172.865,32.786,156.074
C07902=1060.985,232.239,409.697,172.863,32.781,156.073
C07903=1060.979,231.992,409.724,172.860,32.778,156.072
C07904=1060.973,231.742,409.751,172.858,32.774,156.072
C07905=1060.966,231.495,409.779,172.856,32.770,156.071
C07906=1060.960,231.246,409.806,172.854,32.766,156.070
C07907=1060.954,230.997,409.832,172.851,32.762,156.069
C07908=1060.948,230.749,409.859,172.849,32.758,156.069
C07909=1060.942,230.501,409.887,172.847,32.754,156.068
C07910=1060.936,230.252,409.913,172.845,32.750,156.067
C07911=1060.930,230.003,409.940,172.843,32.747,156.066
C07912=1060.924,229.755,409.967,172.840,32.743,156.066
C07913=1060.918,229.507,409.994,172.838,32.739,156.065
C07914=1060.911,229.258,410.021,172.836,32.735,156.064
C07915=1060.906,229.010,410.048,172.834,32.731,156.063
C07916=1060.899,228.761,410.075,172.832,32.727,156.063
C07917=1060.894,228.512,410.102,172.830,32.723,156.062
C07918=1060.886,228.264,410.129,172.827,32.720,156.061
C07919=1060.880,228.016,410.155,172.825,32.715,156.061
C07920=1060.875,227.767,410.182,172.823,32.712,156.060
C07921=1060.868,227.518,410.209,172.821,32.707,156.059
C07922=1060.862,227.270,410.236,172.819,32.704,156.058
C07923=1060.857,227.022,410.262,172.816,32.700,156.058
C07924=1060.850,226.773,410.289,172.814,32.696,156.057
C07925=1060.844,226.524,410.315,172.812,32.692,156.056
C07926=1060.837,226.275,410.342,172.810,32.688,156.056
C07927=1060.832,226.027,410.369,172.808,32.684,156.055
C07928=1060.826,225.779,410.396,172.806,32.680,156.054
C07929=1060.819,225.530,410.423,172.803,32.676,156.053
C07930=1060.813,225.282,410.449,172.801,32.672,156.053
C07931=1060.807,225.033,410.476,172.799,32.669,156.052
C07932=1060.801,224.784,410.503,172.798,32.664,156.051
C07933=1060.795,224.536,410.529,172.796,32.661,156.050
C07934=1060.789,224.287,410.556,172.794,32.657,156.050
C07935=1060.783,224.039,410.582,172.792,32.653,156.049
C07936=1060.776,223.790,410.609,172.789,32.649,156.048
C07937=1060.771,223.542,410.636,172.787,32.645,156.048
C07938=1060.765,223.294,410.662,172.785,32.641,156.047
C07939=1060.758,223.045,410.689,172.783,32.637,156.046
C07940=1060.752,222.796,410.715,172.781,32.633,156.045
C07941=1060.747,222.565,410.740,172.779,32.630,156.045
C07942=1060.741,222.333,410.765,172.777,32.626,156.044
C07943=1060.735,222.100,410.790,172.775,32.622,156.043
C07944=1060.730,221.868,410.814,172.773,32.618,156.043
C07945=1060.724,221.636,410.839,172.771,32.615,156.042
C07946=1060.718,221.404,410.864,172.769,32.611,156.041
C07947=1060.713,221.172,410.889,172.767,32.607,156.040
C07948=1060.707,220.939,410.913,172.765,32.603,156.040
C07949=1060.701,220.691,410.939,172.763,32.600,156.039
C07950=1060.694,220.442,410.966,172.761,32.596,156.038
C07951=1060.688,220.194,410.992,172.759,32.592,156.038
C07952=1060.682,219.945,411.018,172.757,32.588,156.037
C07953=1060.677,219.697,411.045,172.754,32.584,156.036
C07954=1060.670,219.448,411.071,172.752,32.580,156.035
C07955=1060.664,219.199,411.097,172.750,32.576,156.035
C07956=1060.658,218.951,411.123,172.749,32.572,156.034
C07957=1060.652,218.703,411.150,172.747,32.568,156.033
C07958=1060.645,218.454,411.176,172.745,32.565,156.033
C07959=1060.639,218.205,411.202,172.743,32.560,156.032
C07960=1060.633,217.957,411.228,172.741,32.557,156.031
C07961=1060.627,217.709,411.255,172.739,32.552,156.030
C07962=1060.621,217.460,411.280,172.737,32.549,156.030
C07963=1060.614,217.211,411.307,172.734,32.544,156.029
C07964=1060.608,216.962,411.333,172.732,32.541,156.028
C07965=1060.602,216.714,411.359,172.730,32.536,156.027
C07966=1060.596,216.466,411.385,172.728,32.533,156.027
C07967=1060.590,216.217,411.411,172.726,32.528,156.026
C07968=1060.584,215.969,411.437,172.724,32.525,156.025
C07969=1060.578,215.720,411.463,172.722,32.520,156.024
C07970=1060.571,215.471,411.490,172.720,32.517,156.024
C07971=1060.566,215.222,411.516,172.718,32.512,156.023
C07972=1060.559,214.974,411.542,172.716,32.509,156.022
C07973=1060.554,214.725,411.568,172.714,32.505,156.021
C07974=1060.547,214.477,411.594,172.712,32.501,156.021
C07975=1060.542,214.228,411.620,172.711,32.497,156.020
C07976=1060.535,213.980,411.646,172.709,32.493,156.019
C07977=1060.530,213.731,411.671,172.707,32.489,156.019
C07978=1060.523,213.483,411.698,172.704,32.485,156.018
C07979=1060.518,213.234,411.723,172.702,32.481,156.017
C07980=1060.511,212.985,411.750,172.700,32.477,156.016
C07981=1060.505,212.737,411.775,172.698,32.473,156.016
C07982=1060.499,212.488,411.802,172.696,32.469,156.015
C07983=1060.493,212.240,411.827,172.694,32.465,156.014
C07984=1060.486,211.991,411.853,172.692,32.461,156.013
C07985=1060.481,211.743,411.879,172.690,32.457,156.013
C07986=1060.474,211.494,411.905,172.688,32.453,156.012
C07987=1060.468,211.245,411.930,172.686,32.449,156.011
C07988=1060.462,210.997,411.957,172.684,32.445,156.010
C07989=1060.456,210.748,411.982,172.682,32.441,156.010
C07990=1060.450,210.500,412.007,172.681,32.437,156.009
C07991=1060.444,210.251,412.034,172.679,32.433,156.008
C07992=1060.438,210.002,412.059,172.677,32.428,156.007
C07993=1060.432,209.754,412.085,172.675,32.425,156.007
C07994=1060.426,209.505,412.110,172.673,32.420,156.006
C07995=1060.420,209.257,412.137,172.671,32.417,156.005
C07996=1060.414,209.008,412.162,172.669,32.413,156.004
C07997=1060.408,208.778,412.185,172.667,32.409,156.004
C07998=1060.403,208.549,412.209,172.665,32.405,156.003
C07999=1060.396,208.319,412.233,172.663,32.401,156.002
C08000=1060.391,208.090,412.256,172.661,32.398,156.002
C08001=1060.385,207.860,412.280,172.660,32.394,156.001
C08002=1060.380,207.630,412.303,172.658,32.390,156.000
C08003=1060.373,207.401,412.327,172.656,32.387,156.000
C08004=1060.368,207.170,412.351,172.654,32.383,155.999
C08005=1060.344,206.122,412.455,172.475,32.298,155.990
C08006=1060.337,205.873,412.480,172.472,32.295,155.989
C08007=1060.331,205.625,412.504,172.470,32.292,155.989
C08008=1060.325,205.375,412.529,172.468,32.289,155.988
C08009=1060.319,205.127,412.554,172.465,32.286,155.988
C08010=1060.314,204.878,412.578,172.463,32.282,155.987
C08011=1060.308,204.629,412.604,172.460,32.279,155.987
C08012=1060.302,204.381,412.628,172.458,32.276,155.986
C08013=1060.296,204.132,412.652,172.456,32.273,155.985
C08014=1060.290,203.884,412.677,172.453,32.270,155.985
C08015=1060.284,203.635,412.701,172.451,32.267,155.984
C08016=1060.279,203.386,412.726,172.449,32.263,155.984
C08017=1060.273,203.137,412.750,172.447,32.261,155.983
C08018=1060.267,202.889,412.775,172.445,32.258,155.983
C08019=1060.262,202.639,412.800,172.443,32.254,155.982
C08020=1060.256,202.391,412.824,172.440,32.251,155.982
C08021=1060.249,202.142,412.849,172.438,32.248,155.981
C08022=1060.243,201.893,412.874,172.436,32.245,155.981
C08023=1060.238,201.645,412.898,172.433,32.242,155.980
C08024=1060.231,201.396,412.922,172.431,32.239,155.980
C08025=1060.226,201.147,412.946,172.428,32.236,155.979
C08026=1060.220,200.898,412.970,172.426,32.233,155.979
C08027=1060.214,200.650,412.995,172.424,32.230,155.978
C08028=1060.207,200.401,413.019,172.422,32.227,155.978
C08029=1060.202,200.153,413.043,172.420,32.224,155.977
C08030=1060.195,199.904,413.067,172.418,32.220,155.977
C08031=1060.190,199.655,413.092,172.415,32.218,155.976
C08032=1060.184,199.406,413.116,172.413,32.215,155.976
C08033=1060.178,199.157,413.140,172.411,32.211,155.975
C08034=1060.172,198.908,413.165,172.408,32.209,155.975
C08035=1060.166,198.660,413.188,172.406,32.205,155.974
C08036=1060.160,198.411,413.213,172.404,32.202,155.974
C08037=1060.154,198.162,413.236,172.401,32.199,155.973
C08038=1060.148,197.913,413.261,172.399,32.196,155.973
C08039=1060.142,197.665,413.285,172.397,32.193,155.972
C08040=1060.136,197.415,413.309,172.395,32.190,155.971
C08041=1060.130,197.167,413.333,172.393,32.187,155.971
C08042=1060.124,196.918,413.358,172.391,32.184,155.970
C08043=1060.118,196.670,413.381,172.388,32.181,155.970
C08044=1060.113,196.420,413.406,172.386,32.178,155.970
C08045=1060.106,196.172,413.430,172.384,32.175,155.969
C08046=1060.101,195.923,413.454,172.382,32.172,155.968
C08047=1060.095,195.674,413.478,172.379,32.169,155.968
C08048=1060.089,195.426,413.502,172.377,32.166,155.967
C08049=1060.083,195.177,413.526,172.375,32.163,155.967
C08050=1060.077,194.928,413.550,172.373,32.160,155.967
C08051=1060.071,194.680,413.574,172.371,32.157,155.966
C08052=1060.066,194.430,413.598,172.369,32.154,155.965
C08053=1060.060,194.182,413.622,172.366,32.151,155.965
C08054=1060.054,193.933,413.646,172.364,32.148,155.964
C08055=1060.048,193.684,413.670,172.362,32.145,155.964
C08056=1060.042,193.436,413.694,172.360,32.142,155.963
C08057=1060.036,193.187,413.718,172.357,32.139,155.963
C08058=1060.031,192.937,413.742,172.355,32.136,155.962
C08059=1060.025,192.689,413.765,172.353,32.133,155.962
C08060=1060.019,192.440,413.790,172.351,32.130,155.961
C08061=1060.013,192.192,413.814,172.349,32.127,155.961
C08062=1060.007,191.943,413.837,172.347,32.124,155.960
C08063=1060.002,191.694,413.861,172.345,32.121,155.960
C08064=1059.995,191.445,413.885,172.343,32.118,155.959
C08065=1059.990,191.197,413.909,172.340,32.115,155.959
C08066=1059.982,190.878,413.940,172.337,32.111,155.958
C08067=1059.975,190.558,413.971,172.335,32.108,155.958
C08068=1059.967,190.240,414.001,172.332,32.104,155.957
C08069=1059.960,189.920,414.030,172.329,32.100,155.956
C08070=1059.955,189.671,414.055,172.328,32.097,155.956
C08071=1059.948,189.423,414.079,172.325,32.094,155.955
C08072=1059.943,189.173,414.102,172.323,32.091,155.955
C08073=1059.937,188.925,414.126,172.321,32.088,155.954
C08074=1059.932,188.676,414.150,172.319,32.085,155.954
C08075=1059.925,188.427,414.174,172.316,32.082,155.953
C08076=1059.919,188.179,414.197,172.314,32.079,155.953
C08077=1059.914,187.930,414.221,172.312,32.076,155.952
C08078=1059.908,187.681,414.244,172.310,32.073,155.952
C08079=1059.903,187.432,414.269,172.307,32.070,155.951
C08080=1059.897,187.183,414.292,172.306,32.067,155.951
C08081=1059.891,186.935,414.316,172.304,32.064,155.950
C08082=1059.886,186.685,414.339,172.302,32.061,155.950
C08083=1059.879,186.437,414.363,172.300,32.058,155.949
C08084=1059.874,186.188,414.386,172.297,32.055,155.949
C08085=1059.868,185.939,414.410,172.295,32.052,155.948
C08086=1059.862,185.690,414.433,172.293,32.049,155.948
C08087=1059.857,185.441,414.458,172.291,32.046,155.947
C08088=1059.851,185.193,414.481,172.289,32.043,155.947
C08089=1059.846,184.944,414.505,172.286,32.040,155.946
C08090=1059.840,184.695,414.528,172.285,32.037,155.946
C08091=1059.834,184.447,414.551,172.283,32.034,155.945
C08092=1059.828,184.197,414.575,172.281,32.032,155.945
C08093=1059.822,183.948,414.598,172.279,32.028,155.944
C08094=1059.816,183.700,414.621,172.276,32.026,155.944
C08095=1059.810,183.450,414.645,172.274,32.023,155.944
C08096=1059.804,183.202,414.668,172.272,32.020,155.943
C08097=1059.798,182.953,414.691,172.270,32.017,155.943
C08098=1059.792,182.704,414.714,172.268,32.015,155.942
C08099=1059.786,182.455,414.738,172.265,32.012,155.942
C08100=1059.780,182.206,414.761,172.264,32.009,155.941
C08101=1059.774,181.958,414.784,172.262,32.006,155.941
C08102=1059.768,181.709,414.806,172.260,32.003,155.940
C08103=1059.761,181.461,414.830,172.258,32.001,155.940
C08104=1059.755,181.211,414.853,172.255,31.998,155.939
C08105=1059.749,180.962,414.876,172.253,31.995,155.939
C08106=1059.744,180.713,414.899,172.251,31.992,155.938
C08107=1059.738,180.464,414.922,172.249,31.989,155.938
C08108=1059.732,180.216,414.946,172.247,31.986,155.937
C08109=1059.726,179.967,414.969,172.246,31.984,155.937
C08110=1059.720,179.718,414.992,172.243,31.981,155.937
C08111=1059.713,179.469,415.015,172.241,31.978,155.936
C08112=1059.708,179.220,415.037,172.239,31.975,155.936
C08113=1059.702,178.972,415.061,172.237,31.973,155.935
C08114=1059.696,178.723,415.084,172.235,31.970,155.935
C08115=1059.690,178.474,415.107,172.233,31.967,155.934
C08116=1059.684,178.225,415.130,172.230,31.964,155.934
C08117=1059.678,177.976,415.153,172.228,31.961,155.933
C08118=1059.672,177.727,415.176,172.226,31.958,155.933
C08119=1059.666,177.478,415.199,172.225,31.956,155.932
C08120=1059.660,177.229,415.222,172.223,31.953,155.932
C08121=1059.654,176.981,415.245,172.221,31.950,155.931
C08122=1059.648,176.732,415.268,172.218,31.947,155.931
C08123=1059.643,176.483,415.291,172.216,31.945,155.931
C08124=1059.637,176.234,415.314,172.214,31.941,155.930
C08125=1059.630,175.985,415.337,172.212,31.939,155.930
C08126=1059.626,175.771,415.356,172.210,31.936,155.929
C08127=1059.620,175.558,415.376,172.208,31.934,155.929
C08128=1059.615,175.345,415.395,172.208,31.932,155.928
C08129=1059.610,175.132,415.416,172.206,31.929,155.928
C08130=1059.604,174.847,415.441,172.203,31.926,155.927
C08131=1059.597,174.564,415.467,172.201,31.923,155.927
C08132=1059.590,174.280,415.493,172.198,31.919,155.926
C08133=1059.583,173.996,415.519,172.196,31.917,155.926
C08134=1059.577,173.747,415.542,172.194,31.914,155.925
C08135=1059.571,173.498,415.565,172.192,31.911,155.925
C08136=1059.566,173.249,415.588,172.190,31.908,155.925
C08137=1059.560,173.000,415.611,172.189,31.905,155.924
C08138=1059.554,172.751,415.633,172.186,31.902,155.924
C08139=1059.548,172.502,415.656,172.184,31.900,155.923
C08140=1059.542,172.253,415.679,172.182,31.897,155.923
C08141=1059.537,172.004,415.702,172.180,31.894,155.922
C08142=1059.531,171.755,415.725,172.178,31.891,155.922
C08143=1059.524,171.507,415.747,172.176,31.888,155.921
C08144=1059.519,171.258,415.770,172.174,31.886,155.921
C08145=1059.513,171.009,415.793,172.172,31.883,155.920
C08146=1059.508,170.760,415.815,172.171,31.880,155.920
C08147=1059.502,170.511,415.838,172.169,31.877,155.919
C08148=1059.496,170.263,415.860,172.166,31.874,155.919
C08149=1059.490,170.014,415.883,172.164,31.871,155.918
C08150=1059.484,169.765,415.906,172.162,31.869,155.918
C08151=1059.479,169.515,415.928,172.160,31.866,155.918
C08152=1059.473,169.267,415.951,172.158,31.863,155.917
C08153=1059.467,169.018,415.974,172.156,31.860,155.917
C08154=1059.461,168.769,415.996,172.154,31.858,155.916
C08155=1059.456,168.520,416.019,172.153,31.855,155.916
C08156=1059.449,168.271,416.041,172.151,31.852,155.915
C08157=1059.443,168.022,416.064,172.149,31.849,155.915
C08158=1059.438,167.773,416.087,172.147,31.847,155.914
C08159=1059.433,167.524,416.109,172.145,31.843,155.914
C08160=1059.426,167.276,416.131,172.143,31.841,155.913
C08161=1059.421,167.027,416.154,172.141,31.838,155.913
C08162=1059.415,166.777,416.176,172.138,31.835,155.913
C08163=1059.410,166.528,416.199,172.137,31.832,155.912
C08164=1059.403,166.280,416.222,172.135,31.830,155.912
C08165=1059.398,166.030,416.244,172.133,31.826,155.911
C08166=1059.392,165.782,416.266,172.131,31.824,155.911
C08167=1059.387,165.533,416.289,172.129,31.821,155.910
C08168=1059.381,165.284,416.311,172.127,31.818,155.910
C08169=1059.375,165.035,416.334,172.125,31.815,155.909
C08170=1059.369,164.786,416.357,172.123,31.813,155.909
C08171=1059.363,164.537,416.379,172.121,31.810,155.908
C08172=1059.358,164.289,416.401,172.120,31.807,155.908
C08173=1059.352,164.039,416.423,172.118,31.804,155.907
C08174=1059.347,163.790,416.446,172.116,31.801,155.907
C08175=1059.341,163.541,416.468,172.114,31.799,155.907
C08176=1059.335,163.292,416.491,172.112,31.796,155.906
C08177=1059.330,163.044,416.513,172.110,31.793,155.906
C08178=1059.324,162.795,416.535,172.108,31.790,155.905
C08179=1059.318,162.546,416.558,172.106,31.788,155.905
C08180=1059.312,162.297,416.580,172.105,31.785,155.904
C08181=1059.306,162.049,416.602,172.103,31.782,155.904
C08182=1059.301,161.799,416.624,172.101,31.779,155.903
C08183=1059.295,161.550,416.647,172.099,31.776,155.903
C08184=1059.290,161.301,416.670,172.097,31.773,155.902
C08185=1059.284,161.053,416.692,172.095,31.771,155.902
C08186=1059.279,160.803,416.714,172.093,31.768,155.902
C08187=1059.272,160.554,416.736,172.091,31.765,155.901
C08188=1059.266,160.306,416.758,172.090,31.762,155.901
C08189=1059.261,160.056,416.780,172.088,31.760,155.900
C08190=1059.255,159.808,416.802,172.086,31.757,155.900
C08191=1059.249,159.559,416.824,172.084,31.754,155.899
C08192=1059.243,159.309,416.846,172.082,31.752,155.899
C08193=1059.237,159.061,416.868,172.080,31.749,155.898
C08194=1059.231,158.776,416.893,172.077,31.746,155.898
C08195=1059.224,158.492,416.919,172.075,31.743,155.897
C08196=1059.216,158.207,416.943,172.074,31.740,155.897
C08197=1059.210,157.923,416.968,172.071,31.737,155.896
C08198=1059.204,157.674,416.990,172.069,31.734,155.896
C08199=1059.198,157.425,417.013,172.067,31.731,155.896
C08200=1059.192,157.176,417.034,172.065,31.729,155.895
C08201=1059.187,156.928,417.056,172.063,31.726,155.895
C08202=1059.181,156.678,417.078,172.061,31.723,155.894
C08203=1059.175,156.430,417.100,172.059,31.720,155.894
C08204=1059.168,156.180,417.122,172.058,31.718,155.893
C08205=1059.164,155.932,417.144,172.056,31.715,155.893
C08206=1059.158,155.682,417.165,172.054,31.712,155.893
C08207=1059.151,155.433,417.187,172.052,31.710,155.892
C08208=1059.146,155.185,417.210,172.050,31.707,155.892
C08209=1059.140,154.936,417.231,172.048,31.704,155.891
C08210=1059.134,154.687,417.253,172.046,31.701,155.891
C08211=1059.128,154.437,417.275,172.044,31.699,155.890
C08212=1059.122,154.189,417.296,172.044,31.696,155.890
C08213=1059.117,153.939,417.318,172.042,31.694,155.889
C08214=1059.110,153.691,417.340,172.040,31.691,155.889
C08215=1059.104,153.442,417.362,172.038,31.688,155.889
C08216=1059.099,153.193,417.383,172.036,31.686,155.888
C08217=1059.092,152.944,417.405,172.034,31.683,155.888
C08218=1059.086,152.695,417.427,172.032,31.681,155.887
C08219=1059.081,152.446,417.448,172.030,31.677,155.887
C08220=1059.075,152.197,417.470,172.029,31.675,155.886
C08221=1059.069,151.947,417.492,172.027,31.672,155.886
C08222=1059.064,151.699,417.513,172.025,31.669,155.886
C08223=1059.057,151.450,417.535,172.023,31.667,155.885
C08224=1059.051,151.200,417.556,172.021,31.664,155.885
C08225=1059.046,150.952,417.578,172.019,31.662,155.884
C08226=1059.040,150.702,417.600,172.017,31.659,155.884
C08227=1059.034,150.453,417.621,172.015,31.656,155.883
C08228=1059.028,150.205,417.643,172.014,31.654,155.883
C08229=1059.022,149.956,417.664,172.012,31.651,155.883
C08230=1059.016,149.706,417.686,172.010,31.648,155.882
C08231=1059.011,149.458,417.707,172.008,31.645,155.882
C08232=1059.004,149.209,417.729,172.006,31.643,155.881
C08233=1058.998,148.959,417.750,172.004,31.640,155.881
C08234=1058.993,148.711,417.772,172.002,31.637,155.880
C08235=1058.987,148.461,417.794,172.000,31.635,155.880
C08236=1058.982,148.213,417.815,171.999,31.632,155.880
C08237=1058.976,147.964,417.837,171.997,31.629,155.879
C08238=1058.969,147.714,417.859,171.996,31.627,155.879
C08239=1058.964,147.466,417.880,171.994,31.624,155.878
C08240=1058.958,147.217,417.901,171.992,31.622,155.878
C08241=1058.951,146.968,417.923,171.990,31.619,155.877
C08242=1058.946,146.718,417.944,171.988,31.616,155.877
C08243=1058.939,146.470,417.965,171.986,31.614,155.877
C08244=1058.934,146.221,417.986,171.985,31.611,155.876
C08245=1058.928,145.972,418.008,171.983,31.609,155.876
C08246=1058.921,145.723,418.029,171.981,31.606,155.875
C08247=1058.916,145.473,418.050,171.979,31.603,155.875
C08248=1058.910,145.224,418.071,171.977,31.601,155.874
C08249=1058.904,144.976,418.093,171.975,31.598,155.874
C08250=1058.898,144.727,418.114,171.973,31.595,155.874
C08251=1058.892,144.477,418.136,171.972,31.593,155.873
C08252=1058.887,144.228,418.156,171.970,31.590,155.873
C08253=1058.881,143.979,418.178,171.968,31.588,155.872
C08254=1058.875,143.731,418.199,171.967,31.585,155.872
C08255=1058.868,143.482,418.220,171.965,31.582,155.871
C08256=1058.863,143.233,418.241,171.963,31.580,155.871
C08257=1058.857,142.983,418.263,171.961,31.577,155.871
C08258=1058.851,142.699,418.287,171.959,31.574,155.870
C08259=1058.844,142.414,418.312,171.957,31.571,155.870
C08260=1058.837,142.129,418.335,171.955,31.568,155.869
C08261=1058.830,141.845,418.359,171.953,31.565,155.869
C08262=1058.824,141.596,418.381,171.951,31.563,155.868
C08263=1058.818,141.346,418.401,171.949,31.560,155.868
C08264=1058.813,141.098,418.423,171.947,31.557,155.867
C08265=1058.807,140.849,418.444,171.945,31.555,155.867
C08266=1058.801,140.600,418.465,171.945,31.552,155.867
C08267=1058.795,140.350,418.487,171.943,31.549,155.866
C08268=1058.790,140.102,418.508,171.941,31.546,155.866
C08269=1058.783,139.852,418.528,171.939,31.544,155.865
C08270=1058.778,139.604,418.549,171.937,31.542,155.865
C08271=1058.772,139.354,418.570,171.935,31.539,155.865
C08272=1058.766,139.105,418.592,171.933,31.536,155.864
C08273=1058.760,138.856,418.612,171.932,31.534,155.864
C08274=1058.753,138.607,418.634,171.930,31.531,155.863
C08275=1058.748,138.358,418.655,171.928,31.528,155.863
C08276=1058.742,138.109,418.675,171.927,31.526,155.862
C08277=1058.736,137.860,418.696,171.925,31.523,155.862
C08278=1058.730,137.611,418.717,171.923,31.521,155.862
C08279=1058.724,137.362,418.739,171.921,31.518,155.861
C08280=1058.718,137.113,418.759,171.919,31.515,155.861
C08281=1058.712,136.864,418.780,171.918,31.513,155.860
C08282=1058.707,136.615,418.801,171.916,31.510,155.860
C08283=1058.700,136.366,418.822,171.914,31.508,155.859
C08284=1058.695,136.117,418.842,171.912,31.505,155.859
C08285=1058.688,135.867,418.863,171.911,31.502,155.859
C08286=1058.683,135.619,418.884,171.909,31.500,155.858
C08287=1058.677,135.369,418.905,171.907,31.497,155.858
C08288=1058.670,135.121,418.926,171.906,31.494,155.857
C08289=1058.664,134.871,418.946,171.904,31.492,155.857
C08290=1058.659,134.622,418.967,171.902,31.490,155.857
C08291=1058.653,134.374,418.988,171.900,31.487,155.856
C08292=1058.647,134.124,419.009,171.898,31.484,155.856
C08293=1058.642,133.875,419.030,171.897,31.482,155.855
C08294=1058.635,133.626,419.050,171.895,31.479,155.855
C08295=1058.630,133.377,419.071,171.894,31.477,155.855
C08296=1058.623,133.128,419.091,171.892,31.474,155.854
C08297=1058.618,132.879,419.112,171.890,31.471,155.854
C08298=1058.612,132.629,419.133,171.888,31.469,155.853
C08299=1058.605,132.381,419.154,171.886,31.466,155.853
C08300=1058.600,132.131,419.174,171.885,31.464,155.852
C08301=1058.595,131.882,419.195,171.883,31.461,155.852
C08302=1058.588,131.633,419.216,171.882,31.458,155.852
C08303=1058.582,131.385,419.236,171.880,31.456,155.851
C08304=1058.576,131.135,419.257,171.878,31.453,155.851
C08305=1058.570,130.886,419.277,171.876,31.451,155.850
C08306=1058.565,130.637,419.298,171.874,31.448,155.850
C08307=1058.558,130.388,419.319,171.872,31.446,155.850
C08308=1058.552,130.139,419.338,171.871,31.443,155.849
C08309=1058.546,129.889,419.359,171.870,31.441,155.849
C08310=1058.540,129.641,419.379,171.868,31.438,155.848
C08311=1058.533,129.392,419.400,171.866,31.436,155.848
C08312=1058.528,129.143,419.421,171.864,31.433,155.848
C08313=1058.522,128.894,419.441,171.862,31.431,155.847
C08314=1058.515,128.644,419.461,171.860,31.428,155.847
C08315=1058.510,128.395,419.482,171.859,31.425,155.846
C08316=1058.504,128.146,419.502,171.857,31.423,155.846
C08317=1058.497,127.897,419.523,171.856,31.421,155.846
C08318=1058.492,127.648,419.543,171.854,31.418,155.845
C08319=1058.485,127.399,419.564,171.852,31.415,155.845
C08320=1058.479,127.150,419.584,171.850,31.413,155.844
C08321=1058.474,126.901,419.604,171.848,31.410,155.844
C08322=1058.466,126.616,419.627,171.846,31.407,155.844
C08323=1058.460,126.331,419.651,171.845,31.404,155.843
C08324=1058.454,126.046,419.674,171.843,31.402,155.843
C08325=1058.446,125.761,419.697,171.841,31.399,155.842
C08326=1058.441,125.512,419.717,171.839,31.396,155.842
C08327=1058.435,125.263,419.737,171.837,31.394,155.841
C08328=1058.428,125.014,419.758,171.836,31.391,155.841
C08329=1058.423,124.765,419.778,171.834,31.388,155.841
C08330=1058.417,124.516,419.798,171.833,31.386,155.840
C08331=1058.411,124.267,419.818,171.831,31.383,155.840
C08332=1058.404,124.018,419.839,171.829,31.381,155.839
C08333=1058.399,123.768,419.859,171.827,31.378,155.839
C08334=1058.393,123.520,419.879,171.826,31.376,155.839
C08335=1058.386,123.270,419.899,171.824,31.373,155.838
C08336=1058.381,123.021,419.920,171.822,31.371,155.838
C08337=1058.375,122.772,419.940,171.821,31.368,155.837
C08338=1058.369,122.523,419.960,171.819,31.365,155.837
C08339=1058.362,122.274,419.980,171.817,31.363,155.836
C08340=1058.357,122.025,420.001,171.816,31.361,155.836
C08341=1058.351,121.776,420.021,171.814,31.358,155.836
C08342=1058.345,121.527,420.041,171.812,31.355,155.835
C08343=1058.339,121.277,420.062,171.810,31.353,155.835
C08344=1058.333,121.028,420.081,171.809,31.350,155.834
C08345=1058.327,120.780,420.101,171.808,31.348,155.834
C08346=1058.321,120.531,420.121,171.806,31.345,155.834
C08347=1058.316,120.280,420.142,171.804,31.342,155.833
C08348=1058.310,120.032,420.162,171.802,31.340,155.833
C08349=1058.304,119.783,420.182,171.800,31.338,155.833
C08350=1058.298,119.534,420.201,171.799,31.335,155.832
C08351=1058.293,119.285,420.222,171.798,31.332,155.832
C08352=1058.286,119.035,420.242,171.796,31.330,155.831
C08353=1058.280,118.786,420.262,171.794,31.327,155.831
C08354=1058.274,118.537,420.282,171.792,31.324,155.830
C08355=1058.269,118.288,420.302,171.791,31.322,155.830
C08356=1058.263,118.039,420.322,171.789,31.319,155.830
C08357=1058.257,117.790,420.342,171.788,31.317,155.829
C08358=1058.250,117.541,420.362,171.786,31.314,155.829
C08359=1058.245,117.291,420.382,171.784,31.311,155.828
C08360=1058.239,117.042,420.402,171.783,31.309,155.828
C08361=1058.233,116.793,420.422,171.781,31.307,155.828
C08362=1058.228,116.545,420.442,171.779,31.304,155.827
C08363=1058.222,116.295,420.461,171.777,31.301,155.827
C08364=1058.217,116.046,420.482,171.776,31.299,155.826
C08365=1058.210,115.797,420.502,171.775,31.296,155.826
C08366=1058.204,115.548,420.522,171.773,31.294,155.825
C08367=1058.198,115.298,420.541,171.771,31.291,155.825
C08368=1058.193,115.049,420.562,171.769,31.288,155.825
C08369=1058.187,114.800,420.582,171.767,31.286,155.824
C08370=1058.181,114.551,420.601,171.767,31.283,155.824
C08371=1058.175,114.302,420.621,171.765,31.280,155.823
C08372=1058.169,114.053,420.641,171.763,31.278,155.823
C08373=1058.163,113.803,420.661,171.761,31.275,155.823
C08374=1058.157,113.554,420.681,171.760,31.273,155.822
C08375=1058.151,113.306,420.701,171.758,31.271,155.822
C08376=1058.145,113.056,420.720,171.756,31.268,155.821
C08377=1058.139,112.807,420.740,171.755,31.265,155.821
C08378=1058.134,112.558,420.759,171.753,31.263,155.821
C08379=1058.128,112.309,420.779,171.752,31.261,155.820
C08380=1058.122,112.060,420.799,171.750,31.258,155.820
C08381=1058.115,111.810,420.819,171.748,31.255,155.819
C08382=1058.109,111.561,420.839,171.746,31.253,155.819
C08383=1058.104,111.312,420.858,171.746,31.250,155.819
C08384=1058.098,111.063,420.878,171.744,31.247,155.818
C08385=1058.092,110.814,420.897,171.742,31.245,155.818
C08386=1058.085,110.529,420.920,171.740,31.242,155.817
C08387=1058.078,110.244,420.942,171.738,31.239,155.817
C08388=1058.071,109.959,420.964,171.736,31.237,155.817
C08389=1058.065,109.675,420.987,171.735,31.234,155.816
C08390=1058.058,109.425,421.006,171.733,31.231,155.816
C08391=1058.052,109.176,421.026,171.731,31.229,155.815
C08392=1058.046,108.926,421.045,171.729,31.226,155.815
C08393=1058.040,108.678,421.065,171.728,31.224,155.814
C08394=1058.034,108.428,421.084,171.726,31.222,155.814
C08395=1058.029,108.179,421.104,171.724,31.219,155.814
C08396=1058.022,107.930,421.123,171.723,31.216,155.813
C08397=1058.016,107.681,421.142,171.722,31.214,155.813
C08398=1058.010,107.432,421.162,171.720,31.211,155.812
C08399=1058.005,107.183,421.181,171.718,31.209,155.812
C08400=1057.999,106.934,421.201,171.716,31.206,155.812
C08401=1057.992,106.685,421.220,171.714,31.204,155.811
C08402=1057.986,106.435,421.240,171.714,31.201,155.811
C08403=1057.980,106.186,421.260,171.712,31.198,155.811
C08404=1057.974,105.936,421.279,171.710,31.196,155.810
C08405=1057.969,105.687,421.298,171.708,31.194,155.810
C08406=1057.962,105.438,421.317,171.707,31.191,155.809
C08407=1057.956,105.189,421.337,171.705,31.188,155.809
C08408=1057.950,104.940,421.356,171.703,31.186,155.809
C08409=1057.944,104.691,421.376,171.702,31.184,155.808
C08410=1057.939,104.441,421.395,171.701,31.181,155.808
C08411=1057.932,104.192,421.414,171.699,31.179,155.807
C08412=1057.926,103.943,421.434,171.697,31.176,155.807
C08413=1057.921,103.694,421.453,171.695,31.173,155.807
C08414=1057.915,103.444,421.472,171.694,31.171,155.806
C08415=1057.909,103.195,421.491,171.693,31.169,155.806
C08416=1057.903,102.947,421.511,171.691,31.166,155.805
C08417=1057.897,102.697,421.530,171.689,31.163,155.805
C08418=1057.891,102.448,421.549,171.688,31.161,155.805
C08419=1057.885,102.199,421.569,171.686,31.158,155.804
C08420=1057.879,101.950,421.588,171.684,31.156,155.804
C08421=1057.873,101.700,421.607,171.683,31.153,155.803
C08422=1057.867,101.451,421.626,171.682,31.151,155.803
C08423=1057.862,101.202,421.645,171.680,31.148,155.803
C08424=1057.856,100.954,421.665,171.678,31.145,155.802
C08425=1057.850,100.704,421.684,171.676,31.143,155.802
C08426=1057.844,100.455,421.703,171.675,31.141,155.801
C08427=1057.838,100.206,421.722,171.674,31.138,155.801
C08428=1057.832,99.956,421.741,171.672,31.136,155.801
C08429=1057.826,99.707,421.760,171.670,31.133,155.800
C08430=1057.820,99.458,421.779,171.669,31.131,155.800
C08431=1057.813,99.209,421.798,171.667,31.128,155.800
C08432=1057.808,98.960,421.818,171.665,31.126,155.799
C08433=1057.801,98.711,421.836,171.663,31.123,155.799
C08434=1057.795,98.461,421.855,171.663,31.121,155.798
C08435=1057.789,98.212,421.874,171.661,31.118,155.798
C08436=1057.783,97.963,421.893,171.659,31.116,155.798
C08437=1057.777,97.714,421.912,171.657,31.114,155.797
C08438=1057.771,97.464,421.931,171.656,31.111,155.797
C08439=1057.766,97.215,421.950,171.654,31.108,155.796
C08440=1057.759,96.966,421.969,171.653,31.106,155.796
C08441=1057.753,96.716,421.988,171.651,31.104,155.796
C08442=1057.747,96.467,422.007,171.650,31.101,155.795
C08443=1057.741,96.218,422.026,171.648,31.098,155.795
C08444=1057.735,95.968,422.045,171.646,31.096,155.795
C08445=1057.729,95.719,422.064,171.644,31.094,155.794
C08446=1057.723,95.471,422.082,171.644,31.091,155.794
C08447=1057.718,95.221,422.102,171.642,31.088,155.793
C08448=1057.711,94.972,422.120,171.640,31.086,155.793
C08449=1057.706,94.723,422.140,171.638,31.084,155.793
C08450=1057.698,94.438,422.161,171.636,31.081,155.792
C08451=1057.691,94.153,422.183,171.634,31.078,155.792
C08452=1057.685,93.869,422.204,171.633,31.075,155.791
C08453=1057.678,93.583,422.226,171.631,31.072,155.791
C08454=1057.672,93.334,422.244,171.630,31.070,155.790
C08455=1057.666,93.085,422.263,171.628,31.067,155.790
C08456=1057.660,92.835,422.282,171.626,31.064,155.790
C08457=1057.653,92.586,422.301,171.625,31.062,155.789
C08458=1057.648,92.337,422.320,171.624,31.060,155.789
C08459=1057.642,92.088,422.338,171.622,31.057,155.788
C08460=1057.636,91.839,422.358,171.620,31.054,155.788
C08461=1057.630,91.590,422.376,171.619,31.053,155.788
C08462=1057.624,91.340,422.396,171.617,31.050,155.787
C08463=1057.618,91.091,422.414,171.616,31.047,155.787
C08464=1057.613,90.842,422.432,171.614,31.044,155.787
C08465=1057.606,90.593,422.451,171.613,31.042,155.786
C08466=1057.600,90.344,422.470,171.611,31.040,155.786
C08467=1057.594,90.094,422.489,171.609,31.037,155.785
C08468=1057.588,89.844,422.507,171.608,31.035,155.785
C08469=1057.582,89.595,422.526,171.606,31.033,155.785
C08470=1057.575,89.346,422.544,171.605,31.030,155.784
C08471=1057.570,89.098,422.563,171.603,31.027,155.784
C08472=1057.564,88.848,422.582,171.602,31.025,155.784
C08473=1057.558,88.599,422.600,171.600,31.023,155.783
C08474=1057.551,88.350,422.618,171.598,31.020,155.783
C08475=1057.546,88.100,422.638,171.597,31.018,155.782
C08476=1057.539,87.851,422.656,171.596,31.015,155.782
C08477=1057.534,87.602,422.674,171.594,31.013,155.782
C08478=1057.527,87.353,422.692,171.592,31.010,155.781
C08479=1057.521,87.104,422.711,171.590,31.008,155.781
C08480=1057.515,86.854,422.730,171.589,31.005,155.780
C08481=1057.509,86.604,422.748,171.587,31.003,155.780
C08482=1057.503,86.355,422.767,171.586,31.000,155.780
C08483=1057.497,86.106,422.784,171.585,30.998,155.779
C08484=1057.491,85.857,422.804,171.583,30.996,155.779
C08485=1057.485,85.608,422.822,171.581,30.993,155.779
C08486=1057.479,85.358,422.840,171.579,30.990,155.778
C08487=1057.473,85.110,422.859,171.579,30.989,155.778
C08488=1057.467,84.861,422.877,171.577,30.986,155.777
C08489=1057.461,84.610,422.896,171.575,30.983,155.777
C08490=1057.455,84.361,422.914,171.573,30.980,155.777
C08491=1057.449,84.113,422.933,171.572,30.979,155.776
C08492=1057.443,83.863,422.951,171.570,30.976,155.776
C08493=1057.436,83.614,422.969,171.569,30.973,155.776
C08494=1057.430,83.364,422.987,171.568,30.971,155.775
C08495=1057.425,83.116,423.006,171.566,30.969,155.775
C08496=1057.419,82.866,423.025,171.564,30.966,155.774
C08497=1057.413,82.617,423.043,171.562,30.964,155.774
C08498=1057.406,82.368,423.061,171.561,30.961,155.774
C08499=1057.401,82.119,423.079,171.560,30.959,155.773
C08500=1057.395,81.869,423.098,171.558,30.956,155.773
C08501=1057.389,81.619,423.116,171.557,30.954,155.773
C08502=1057.383,81.371,423.134,171.555,30.951,155.772
C08503=1057.377,81.121,423.152,171.553,30.949,155.772
C08504=1057.371,80.872,423.171,171.551,30.946,155.771
C08505=1057.364,80.622,423.189,171.551,30.944,155.771
C08506=1057.359,80.374,423.207,171.549,30.941,155.771
C08507=1057.353,80.124,423.226,171.547,30.939,155.770
C08508=1057.347,79.875,423.244,171.546,30.937,155.770
C08509=1057.341,79.626,423.262,171.544,30.934,155.769
C08510=1057.335,79.377,423.280,171.543,30.931,155.769
C08511=1057.329,79.127,423.298,171.541,30.929,155.769
C08512=1057.323,78.878,423.317,171.540,30.927,155.768
C08513=1057.317,78.629,423.335,171.538,30.924,155.768
C08514=1057.311,78.344,423.356,171.536,30.921,155.768
C08515=1057.304,78.058,423.376,171.534,30.918,155.767
C08516=1057.296,77.774,423.398,171.533,30.915,155.767
C08517=1057.289,77.489,423.418,171.531,30.913,155.766
C08518=1057.283,77.239,423.436,171.529,30.910,155.766
C08519=1057.278,76.990,423.453,171.528,30.908,155.765
C08520=1057.271,76.741,423.472,171.526,30.905,155.765
C08521=1057.265,76.492,423.490,171.525,30.903,155.765
C08522=1057.260,76.243,423.508,171.524,30.901,155.764
C08523=1057.253,75.993,423.526,171.522,30.898,155.764
C08524=1057.247,75.744,423.544,171.520,30.896,155.764
C08525=1057.242,75.495,423.562,171.518,30.893,155.763
C08526=1057.235,75.246,423.580,171.517,30.891,155.763
C08527=1057.228,74.996,423.598,171.516,30.888,155.763
C08528=1057.223,74.747,423.615,171.514,30.886,155.762
C08529=1057.216,74.498,423.634,171.513,30.884,155.762
C08530=1057.210,74.248,423.652,171.511,30.881,155.761
C08531=1057.205,73.999,423.669,171.509,30.878,155.761
C08532=1057.199,73.749,423.687,171.507,30.876,155.761
C08533=1057.192,73.500,423.706,171.507,30.874,155.760
C08534=1057.187,73.251,423.724,171.505,30.871,155.760
C08535=1057.180,73.001,423.741,171.503,30.869,155.760
C08536=1057.175,72.752,423.759,171.502,30.866,155.759
C08537=1057.168,72.504,423.777,171.500,30.864,155.759
C08538=1057.162,72.254,423.795,171.499,30.862,155.758
C08539=1057.156,72.005,423.813,171.497,30.859,155.758
C08540=1057.150,71.755,423.831,171.496,30.856,155.758
C08541=1057.144,71.507,423.849,171.494,30.854,155.757
C08542=1057.138,71.257,423.867,171.492,30.852,155.757
C08543=1057.133,71.008,423.884,171.491,30.849,155.756
C08544=1057.126,70.758,423.902,171.490,30.847,155.756
C08545=1057.120,70.509,423.920,171.488,30.844,155.756
C08546=1057.114,70.260,423.937,171.486,30.842,155.755
C08547=1057.108,70.010,423.955,171.485,30.840,155.755
C08548=1057.102,69.762,423.973,171.483,30.837,155.755
C08549=1057.096,69.512,423.991,171.482,30.835,155.754
C08550=1057.090,69.263,424.008,171.481,30.832,155.754
C08551=1057.084,69.013,424.026,171.479,30.830,155.754
C08552=1057.078,68.764,424.044,171.477,30.827,155.753
C08553=1057.072,68.515,424.062,171.476,30.825,155.753
C08554=1057.065,68.265,424.079,171.474,30.822,155.752
C08555=1057.060,68.016,424.097,171.473,30.820,155.752
C08556=1057.054,67.766,424.115,171.471,30.817,155.752
C08557=1057.047,67.518,424.132,171.470,30.815,155.751
C08558=1057.041,67.268,424.149,171.468,30.813,155.751
C08559=1057.036,67.019,424.167,171.466,30.810,155.751
C08560=1057.029,66.770,424.186,171.465,30.808,155.750
C08561=1057.022,66.520,424.203,171.464,30.805,155.750
C08562=1057.017,66.271,424.221,171.462,30.803,155.750
C08563=1057.011,66.021,424.238,171.460,30.801,155.749
C08564=1057.004,65.773,424.255,171.459,30.798,155.749
C08565=1056.998,65.523,424.273,171.457,30.796,155.748
C08566=1056.993,65.274,424.291,171.456,30.793,155.748
C08567=1056.986,65.025,424.308,171.455,30.791,155.748
C08568=1056.981,64.775,424.325,171.453,30.789,155.747
C08569=1056.975,64.525,424.343,171.451,30.786,155.747
C08570=1056.968,64.276,424.360,171.449,30.784,155.747
C08571=1056.962,64.027,424.378,171.449,30.781,155.746
C08572=1056.956,63.778,424.395,171.447,30.779,155.746
C08573=1056.950,63.528,424.413,171.445,30.776,155.746
C08574=1056.944,63.279,424.430,171.444,30.774,155.745
C08575=1056.937,63.030,424.447,171.442,30.772,155.745
C08576=1056.931,62.780,424.465,171.440,30.770,155.744
C08577=1056.924,62.532,424.482,171.439,30.768,155.744
C08578=1056.917,62.246,424.502,171.437,30.765,155.744
C08579=1056.910,61.961,424.522,171.435,30.762,155.743
C08580=1056.904,61.676,424.541,171.433,30.759,155.743
C08581=1056.896,61.391,424.561,171.431,30.757,155.743
C08582=1056.890,61.142,424.578,171.431,30.754,155.742
C08583=1056.884,60.892,424.596,171.429,30.752,155.742
C08584=1056.878,60.643,424.613,171.427,30.749,155.741
C08585=1056.871,60.394,424.631,171.426,30.747,155.741
C08586=1056.866,60.145,424.648,171.424,30.745,155.741
C08587=1056.859,59.895,424.665,171.423,30.743,155.740
C08588=1056.853,59.646,424.682,171.421,30.740,155.740
C08589=1056.847,59.396,424.700,171.420,30.738,155.740
C08590=1056.840,59.147,424.717,171.418,30.735,155.739
C08591=1056.835,58.897,424.734,171.416,30.733,155.739
C08592=1056.828,58.648,424.751,171.415,30.731,155.739
C08593=1056.822,58.399,424.768,171.414,30.728,155.738
C08594=1056.816,58.150,424.786,171.412,30.726,155.738
C08595=1056.810,57.900,424.802,171.410,30.724,155.738
C08596=1056.804,57.651,424.820,171.409,30.721,155.737
C08597=1056.798,57.402,424.837,171.407,30.719,155.737
C08598=1056.791,57.153,424.854,171.406,30.716,155.737
C08599=1056.786,56.903,424.871,171.405,30.714,155.736
C08600=1056.779,56.653,424.888,171.403,30.712,155.736
C08601=1056.772,56.405,424.905,171.401,30.709,155.736
C08602=1056.767,56.155,424.922,171.399,30.707,155.735
C08603=1056.760,55.906,424.940,171.398,30.705,155.735
C08604=1056.755,55.657,424.957,171.397,30.702,155.734
C08605=1056.748,55.407,424.974,171.395,30.700,155.734
C08606=1056.742,55.158,424.991,171.394,30.697,155.734
C08607=1056.737,54.909,425.008,171.392,30.695,155.733
C08608=1056.730,54.659,425.025,171.390,30.693,155.733
C08609=1056.724,54.410,425.042,171.389,30.690,155.733
C08610=1056.718,54.160,425.059,171.388,30.688,155.732
C08611=1056.712,53.911,425.076,171.386,30.685,155.732
C08612=1056.705,53.662,425.093,171.384,30.683,155.732
C08613=1056.700,53.412,425.110,171.382,30.680,155.731
C08614=1056.693,53.163,425.127,171.382,30.678,155.731
C08615=1056.687,52.914,425.143,171.380,30.676,155.730
C08616=1056.681,52.664,425.161,171.378,30.674,155.730
C08617=1056.675,52.415,425.178,171.377,30.671,155.730
C08618=1056.669,52.166,425.195,171.375,30.669,155.729
C08619=1056.663,51.916,425.213,171.374,30.666,155.729
C08620=1056.657,51.667,425.229,171.372,30.664,155.729
C08621=1056.651,51.418,425.246,171.371,30.661,155.728
C08622=1056.645,51.168,425.263,171.369,30.659,155.728
C08623=1056.639,50.919,425.280,171.367,30.657,155.728
C08624=1056.633,50.670,425.296,171.366,30.654,155.727
C08625=1056.627,50.420,425.314,171.365,30.652,155.727
C08626=1056.621,50.171,425.330,171.363,30.649,155.727
C08627=1056.614,49.922,425.347,171.362,30.647,155.726
C08628=1056.609,49.671,425.365,171.360,30.645,155.726
C08629=1056.602,49.423,425.382,171.358,30.642,155.726
C08630=1056.596,49.173,425.398,171.357,30.640,155.725
C08631=1056.591,48.924,425.415,171.356,30.638,155.725
C08632=1056.584,48.674,425.432,171.354,30.635,155.724
C08633=1056.578,48.425,425.448,171.352,30.632,155.724
C08634=1056.573,48.176,425.466,171.351,30.630,155.724
C08635=1056.567,47.927,425.482,171.350,30.628,155.723
C08636=1056.560,47.677,425.499,171.348,30.626,155.723
C08637=1056.555,47.427,425.516,171.346,30.623,155.723
C08638=1056.549,47.179,425.533,171.345,30.621,155.722
C08639=1056.543,46.929,425.550,171.343,30.618,155.722
C08640=1056.536,46.679,425.566,171.342,30.616,155.722
C08641=1056.531,46.430,425.584,171.341,30.613,155.721
C08642=1056.524,46.145,425.602,171.339,30.611,155.721
C08643=1056.517,45.860,425.622,171.337,30.608,155.720
C08644=1056.510,45.574,425.641,171.335,30.605,155.720
C08645=1056.503,45.289,425.660,171.334,30.603,155.720
C08646=1056.497,45.039,425.677,171.332,30.600,155.719
C08647=1056.491,44.790,425.693,171.330,30.597,155.719
C08648=1056.485,44.541,425.710,171.329,30.595,155.719
C08649=1056.479,44.291,425.727,171.327,30.592,155.718
C08650=1056.473,44.042,425.743,171.326,30.590,155.718
C08651=1056.467,43.793,425.760,171.324,30.588,155.717
C08652=1056.461,43.543,425.777,171.323,30.586,155.717
C08653=1056.455,43.294,425.793,171.321,30.583,155.717
C08654=1056.449,43.044,425.810,171.319,30.581,155.716
C08655=1056.442,42.795,425.827,171.319,30.578,155.716
C08656=1056.436,42.546,425.843,171.317,30.576,155.716
C08657=1056.431,42.296,425.860,171.315,30.573,155.715
C08658=1056.425,42.047,425.876,171.313,30.571,155.715
C08659=1056.418,41.798,425.893,171.312,30.569,155.715
C08660=1056.412,41.548,425.910,171.311,30.567,155.714
C08661=1056.407,41.299,425.926,171.309,30.564,155.714
C08662=1056.401,41.050,425.942,171.307,30.562,155.714
C08663=1056.395,40.800,425.958,171.306,30.560,155.713
C08664=1056.388,40.551,425.976,171.304,30.557,155.713
C08665=1056.382,40.301,425.992,171.303,30.555,155.713
C08666=1056.376,40.052,426.008,171.302,30.552,155.712
C08667=1056.370,39.803,426.024,171.300,30.550,155.712
C08668=1056.364,39.553,426.041,171.298,30.548,155.712
C08669=1056.357,39.303,426.057,171.296,30.545,155.711
C08670=1056.351,39.054,426.074,171.296,30.543,155.711
C08671=1056.345,38.805,426.090,171.294,30.541,155.711
C08672=1056.339,38.556,426.107,171.292,30.539,155.710
C08673=1056.333,38.307,426.123,171.290,30.536,155.710
C08674=1056.327,38.057,426.139,171.289,30.534,155.710
C08675=1056.321,37.808,426.156,171.288,30.531,155.709
C08676=1056.315,37.558,426.172,171.286,30.529,155.709
C08677=1056.309,37.308,426.188,171.285,30.527,155.709
C08678=1056.303,37.059,426.205,171.283,30.524,155.708
C08679=1056.297,36.810,426.221,171.281,30.522,155.708
C08680=1056.290,36.561,426.237,171.280,30.519,155.707
C08681=1056.284,36.311,426.253,171.279,30.518,155.707
C08682=1056.278,36.061,426.269,171.277,30.515,155.707
C08683=1056.272,35.812,426.286,171.275,30.513,155.706
C08684=1056.266,35.563,426.302,171.273,30.511,155.706
C08685=1056.259,35.314,426.318,171.272,30.509,155.706
C08686=1056.253,35.064,426.334,171.271,30.506,155.705
C08687=1056.247,34.815,426.350,171.269,30.504,155.705
C08688=1056.241,34.566,426.366,171.267,30.502,155.705
C08689=1056.235,34.315,426.383,171.266,30.499,155.704
C08690=1056.229,34.066,426.399,171.264,30.497,155.704
C08691=1056.222,33.817,426.415,171.263,30.495,155.704
C08692=1056.216,33.568,426.431,171.261,30.492,155.704
C08693=1056.210,33.318,426.447,171.260,30.490,155.703
C08694=1056.204,33.069,426.464,171.258,30.487,155.703
C08695=1056.198,32.820,426.480,171.256,30.485,155.703
C08696=1056.192,32.571,426.496,171.255,30.483,155.702
C08697=1056.186,32.321,426.512,171.254,30.480,155.702
C08698=1056.180,32.071,426.527,171.252,30.478,155.702
C08699=1056.174,31.821,426.544,171.250,30.476,155.701
C08700=1056.167,31.572,426.560,171.248,30.473,155.701
C08701=1056.161,31.323,426.576,171.248,30.472,155.701
C08702=1056.155,31.074,426.592,171.246,30.469,155.700
C08703=1056.149,30.824,426.608,171.244,30.467,155.700
C08704=1056.143,30.575,426.625,171.243,30.465,155.700
C08705=1056.137,30.325,426.640,171.241,30.462,155.699
C08706=1056.130,30.040,426.659,171.240,30.460,155.699
C08707=1056.123,29.755,426.677,171.238,30.457,155.698
C08708=1056.116,29.469,426.695,171.236,30.454,155.698
C08709=1056.109,29.184,426.713,171.234,30.452,155.698
C08710=1056.103,28.934,426.730,171.233,30.449,155.697
C08711=1056.097,28.685,426.745,171.231,30.447,155.697
C08712=1056.091,28.435,426.761,171.230,30.445,155.697
C08713=1056.085,28.186,426.777,171.228,30.443,155.696
C08714=1056.078,27.937,426.793,171.226,30.440,155.696
C08715=1056.072,27.688,426.809,171.225,30.438,155.696
C08716=1056.066,27.438,426.824,171.224,30.436,155.695
C08717=1056.060,27.189,426.840,171.222,30.433,155.695
C08718=1056.054,26.939,426.857,171.220,30.431,155.695
C08719=1056.047,26.690,426.872,171.218,30.429,155.694
C08720=1056.042,26.440,426.888,171.218,30.427,155.694
C08721=1056.035,26.191,426.903,171.216,30.424,155.694
C08722=1056.029,25.942,426.920,171.214,30.422,155.693
C08723=1056.023,25.692,426.935,171.212,30.420,155.693
C08724=1056.017,25.443,426.951,171.210,30.418,155.693
C08725=1056.011,25.194,426.967,171.210,30.415,155.692
C08726=1056.004,24.944,426.982,171.208,30.413,155.692
C08727=1055.998,24.695,426.998,171.206,30.411,155.692
C08728=1055.992,24.445,427.014,171.204,30.408,155.692
C08729=1055.986,24.196,427.030,171.203,30.406,155.691
C08730=1055.980,23.946,427.046,171.202,30.404,155.691
C08731=1055.973,23.697,427.061,171.200,30.402,155.691
C08732=1055.968,23.447,427.077,171.198,30.399,155.690
C08733=1055.961,23.198,427.093,171.197,30.397,155.690
C08734=1055.955,22.948,427.108,171.195,30.395,155.690
C08735=1055.949,22.699,427.124,171.194,30.393,155.689
C08736=1055.943,22.450,427.140,171.192,30.390,155.689
C08737=1055.936,22.200,427.155,171.191,30.388,155.689
C08738=1055.930,21.951,427.171,171.189,30.386,155.688
C08739=1055.924,21.701,427.186,171.187,30.384,155.688
C08740=1055.918,21.452,427.203,171.186,30.381,155.688
C08741=1055.912,21.202,427.218,171.185,30.379,155.687
C08742=1055.906,20.953,427.234,171.183,30.377,155.687
C08743=1055.899,20.703,427.249,171.181,30.374,155.687
C08744=1055.893,20.454,427.265,171.179,30.372,155.686
C08745=1055.888,20.204,427.281,171.178,30.370,155.686
C08746=1055.882,19.955,427.296,171.177,30.368,155.686
C08747=1055.875,19.706,427.311,171.175,30.365,155.685
C08748=1055.869,19.456,427.327,171.173,30.363,155.685
C08749=1055.863,19.207,427.342,171.171,30.361,155.685
C08750=1055.857,18.957,427.358,171.171,30.359,155.685
C08751=1055.851,18.708,427.373,171.169,30.357,155.684
C08752=1055.844,18.459,427.389,171.167,30.354,155.684
C08753=1055.838,18.209,427.404,171.165,30.352,155.684
C08754=1055.832,17.960,427.420,171.164,30.350,155.683
C08755=1055.826,17.710,427.436,171.163,30.348,155.683
C08756=1055.820,17.460,427.451,171.161,30.346,155.683
C08757=1055.813,17.211,427.466,171.159,30.343,155.682
C08758=1055.808,16.962,427.481,171.157,30.341,155.682
C08759=1055.801,16.713,427.497,171.156,30.339,155.682
C08760=1055.795,16.463,427.512,171.155,30.337,155.681
C08761=1055.789,16.213,427.527,171.153,30.335,155.681
C08762=1055.783,15.964,427.543,171.151,30.332,155.681
C08763=1055.777,15.714,427.559,171.150,30.330,155.681
C08764=1055.770,15.464,427.574,171.148,30.328,155.680
C08765=1055.764,15.216,427.589,171.147,30.326,155.680
C08766=1055.759,14.966,427.604,171.145,30.323,155.680
C08767=1055.752,14.717,427.619,171.143,30.321,155.679
C08768=1055.746,14.467,427.635,171.142,30.319,155.679
C08769=1055.740,14.218,427.651,171.140,30.317,155.679
C08770=1055.733,13.933,427.668,171.139,30.314,155.678
C08771=1055.725,13.649,427.685,171.137,30.312,155.678
C08772=1055.719,13.366,427.702,171.135,30.309,155.678
C08773=1055.712,13.081,427.720,171.133,30.307,155.677
C08774=1055.705,12.832,427.735,171.132,30.305,155.677
C08775=1055.699,12.582,427.750,171.130,30.302,155.677
C08776=1055.692,12.333,427.765,171.128,30.300,155.676
C08777=1055.686,12.083,427.780,171.126,30.298,155.676
C08778=1055.680,11.833,427.795,171.125,30.296,155.676
C08779=1055.674,11.585,427.810,171.124,30.294,155.676
C08780=1055.668,11.335,427.826,171.122,30.292,155.675
C08781=1055.661,11.086,427.841,171.120,30.290,155.675
C08782=1055.655,10.836,427.856,171.118,30.288,155.675
C08783=1055.649,10.586,427.871,171.117,30.285,155.674
C08784=1055.642,10.337,427.886,171.116,30.283,155.674
C08785=1055.636,10.088,427.901,171.114,30.281,155.674
C08786=1055.630,9.839,427.916,171.112,30.279,155.674
C08787=1055.623,9.589,427.931,171.110,30.276,155.673
C08788=1055.618,9.339,427.946,171.109,30.274,155.673
C08789=1055.611,9.089,427.961,171.108,30.272,155.673
C08790=1055.606,8.840,427.976,171.106,30.270,155.672
C08791=1055.599,8.591,427.992,171.104,30.268,155.672
C08792=1055.593,8.342,428.007,171.102,30.266,155.672
C08793=1055.586,8.092,428.022,171.101,30.264,155.672
C08794=1055.580,7.842,428.036,171.100,30.262,155.671
C08795=1055.574,7.593,428.051,171.098,30.260,155.671
C08796=1055.568,7.344,428.066,171.096,30.257,155.671
C08797=1055.562,7.094,428.082,171.094,30.255,155.670
C08798=1055.556,6.844,428.096,171.093,30.253,155.670
C08799=1055.550,6.595,428.111,171.092,30.250,155.670
C08800=1055.543,6.345,428.126,171.090,30.248,155.669
C08801=1055.537,6.096,428.141,171.088,30.246,155.669
C08802=1055.531,5.846,428.156,171.086,30.244,155.669
C08803=1055.525,5.597,428.170,171.085,30.242,155.669
C08804=1055.519,5.348,428.185,171.084,30.240,155.668
C08805=1055.512,5.098,428.200,171.082,30.238,155.668
C08806=1055.506,4.849,428.215,171.080,30.236,155.668
C08807=1055.500,4.599,428.230,171.078,30.233,155.667
C08808=1055.494,4.349,428.245,171.076,30.231,155.667
C08809=1055.488,4.100,428.260,171.076,30.229,155.667
C08810=1055.482,3.851,428.275,171.074,30.227,155.667
C08811=1055.476,3.601,428.290,171.072,30.225,155.666
C08812=1055.469,3.351,428.305,171.070,30.223,155.666
C08813=1055.464,3.102,428.319,171.069,30.221,155.666
C08814=1055.457,2.853,428.334,171.068,30.219,155.665
C08815=1055.451,2.603,428.349,171.066,30.217,155.665
C08816=1055.445,2.354,428.364,171.064,30.214,155.665
C08817=1055.439,2.104,428.379,171.062,30.212,155.665
C08818=1055.432,1.855,428.394,171.061,30.209,155.664
C08819=1055.427,1.606,428.408,171.059,30.207,155.664
C08820=1055.420,1.356,428.423,171.058,30.205,155.664
C08821=1055.414,1.107,428.438,171.056,30.203,155.663
C08822=1055.408,0.857,428.452,171.054,30.201,155.663
C08823=1055.402,0.607,428.467,171.053,30.199,155.663
C08824=1055.396,0.358,428.482,171.051,30.197,155.663
C08825=1055.390,0.109,428.497,171.050,30.195,155.662
C08826=1055.383,-0.141,428.512,171.048,30.193,155.662
C08827=1055.378,-0.390,428.526,171.046,30.190,155.662
C08828=1055.371,-0.640,428.541,171.045,30.188,155.661
C08829=1055.366,-0.890,428.556,171.043,30.186,155.661
C08830=1055.360,-1.139,428.570,171.041,30.184,155.661
C08831=1055.354,-1.389,428.585,171.040,30.182,155.661
C08832=1055.348,-1.638,428.600,171.038,30.180,155.660
C08833=1055.342,-1.887,428.615,171.037,30.178,155.660
C08834=1055.334,-2.170,428.630,171.035,30.175,155.660
C08835=1055.328,-2.452,428.647,171.033,30.173,155.659
C08836=1055.321,-2.734,428.664,171.031,30.171,155.659
C08837=1055.314,-3.016,428.680,171.030,30.168,155.659
C08838=1055.308,-3.266,428.695,171.028,30.166,155.658
C08839=1055.302,-3.515,428.710,171.026,30.163,155.658
C08840=1055.296,-3.765,428.724,171.024,30.161,155.658
C08841=1055.289,-4.014,428.738,171.022,30.159,155.658
C08842=1055.283,-4.263,428.753,171.021,30.158,155.657
C08843=1055.277,-4.514,428.767,171.020,30.156,155.657
C08844=1055.271,-4.763,428.782,171.018,30.153,155.657
C08845=1055.264,-5.012,428.796,171.016,30.151,155.656
C08846=1055.258,-5.262,428.811,171.014,30.149,155.656
C08847=1055.252,-5.511,428.825,171.013,30.147,155.656
C08848=1055.246,-5.761,428.840,171.011,30.145,155.656
C08849=1055.239,-6.010,428.853,171.009,30.143,155.655
C08850=1055.233,-6.260,428.868,171.008,30.141,155.655
C08851=1055.227,-6.509,428.883,171.006,30.139,155.655
C08852=1055.220,-6.759,428.896,171.005,30.137,155.655
C08853=1055.214,-7.008,428.911,171.003,30.135,155.654
C08854=1055.209,-7.258,428.925,171.001,30.133,155.654
C08855=1055.202,-7.508,428.940,170.999,30.131,155.654
C08856=1055.196,-7.756,428.954,170.997,30.129,155.654
C08857=1055.190,-8.007,428.968,170.997,30.127,155.653
C08858=1055.183,-8.256,428.983,170.995,30.125,155.653
C08859=1055.177,-8.505,428.997,170.993,30.123,155.653
C08860=1055.171,-8.755,429.012,170.991,30.120,155.653
C08861=1055.165,-9.005,429.025,170.989,30.119,155.652
C08862=1055.158,-9.254,429.040,170.988,30.117,155.652
C08863=1055.153,-9.504,429.054,170.986,30.115,155.652
C08864=1055.146,-9.753,429.069,170.985,30.113,155.651
C08865=1055.141,-10.003,429.082,170.983,30.110,155.651
C08866=1055.134,-10.252,429.097,170.982,30.108,155.651
C08867=1055.128,-10.502,429.111,170.980,30.107,155.651
C08868=1055.122,-10.751,429.126,170.978,30.104,155.651
C08869=1055.115,-11.001,429.139,170.976,30.102,155.650
C08870=1055.109,-11.250,429.154,170.974,30.100,155.650
C08871=1055.104,-11.500,429.168,170.973,30.098,155.650
C08872=1055.096,-11.749,429.182,170.972,30.096,155.649
C08873=1055.091,-11.999,429.196,170.970,30.094,155.649
C08874=1055.085,-12.248,429.211,170.968,30.092,155.649
C08875=1055.078,-12.498,429.224,170.966,30.090,155.649
C08876=1055.072,-12.747,429.239,170.965,30.088,155.648
C08877=1055.067,-12.997,429.253,170.963,30.086,155.648
C08878=1055.060,-13.246,429.266,170.961,30.084,155.648
C08879=1055.054,-13.496,429.281,170.960,30.082,155.648
C08880=1055.048,-13.745,429.295,170.958,30.080,155.647
C08881=1055.041,-13.995,429.309,170.957,30.078,155.647
C08882=1055.036,-14.244,429.323,170.955,30.076,155.647
C08883=1055.029,-14.494,429.337,170.953,30.074,155.647
C08884=1055.023,-14.743,429.351,170.951,30.072,155.646
C08885=1055.017,-14.994,429.366,170.949,30.070,155.646
C08886=1055.011,-15.243,429.379,170.948,30.068,155.646
C08887=1055.005,-15.492,429.394,170.946,30.065,155.646
C08888=1054.998,-15.742,429.407,170.945,30.064,155.645
C08889=1054.993,-15.991,429.421,170.943,30.062,155.645
C08890=1054.986,-16.241,429.435,170.941,30.060,155.645
C08891=1054.980,-16.490,429.449,170.940,30.058,155.645
C08892=1054.973,-16.740,429.463,170.938,30.056,155.644
C08893=1054.967,-16.989,429.477,170.936,30.054,155.644
C08894=1054.961,-17.239,429.491,170.934,30.052,155.644
C08895=1054.955,-17.488,429.504,170.932,30.050,155.644
C08896=1054.949,-17.738,429.518,170.931,30.049,155.644
C08897=1054.942,-17.987,429.533,170.930,30.047,155.643
C08898=1054.936,-18.268,429.548,170.927,30.044,155.643
C08899=1054.928,-18.549,429.563,170.925,30.042,155.643
C08900=1054.921,-18.830,429.579,170.924,30.040,155.642
C08901=1054.915,-19.109,429.595,170.922,30.038,155.642
C08902=1054.908,-19.359,429.609,170.920,30.035,155.642
C08903=1054.902,-19.609,429.622,170.918,30.034,155.642
C08904=1054.896,-19.858,429.636,170.916,30.032,155.641
C08905=1054.889,-20.108,429.649,170.915,30.030,155.641
C08906=1054.884,-20.358,429.663,170.913,30.028,155.641
C08907=1054.877,-20.606,429.677,170.912,30.026,155.641
C08908=1054.870,-20.856,429.691,170.910,30.024,155.640
C08909=1054.865,-21.106,429.705,170.908,30.022,155.640
C08910=1054.858,-21.356,429.718,170.907,30.020,155.640
C08911=1054.853,-21.605,429.732,170.905,30.019,155.640
C08912=1054.846,-21.855,429.745,170.903,30.016,155.640
C08913=1054.840,-22.105,429.759,170.901,30.014,155.639
C08914=1054.834,-22.354,429.774,170.899,30.013,155.639
C08915=1054.828,-22.603,429.787,170.898,30.010,155.639
C08916=1054.822,-22.853,429.801,170.896,30.008,155.639
C08917=1054.815,-23.102,429.814,170.894,30.007,155.638
C08918=1054.809,-23.352,429.828,170.893,30.005,155.638
C08919=1054.804,-23.601,429.842,170.891,30.003,155.638
C08920=1054.797,-23.851,429.855,170.890,30.001,155.638
C08921=1054.791,-24.101,429.869,170.888,29.999,155.637
C08922=1054.785,-24.350,429.882,170.886,29.997,155.637
C08923=1054.778,-24.600,429.896,170.884,29.995,155.637
C08924=1054.772,-24.849,429.909,170.882,29.993,155.637
C08925=1054.767,-25.099,429.923,170.881,29.991,155.637
C08926=1054.760,-25.349,429.937,170.879,29.989,155.636
C08927=1054.754,-25.598,429.951,170.877,29.988,155.636
C08928=1054.748,-25.848,429.964,170.875,29.985,155.636
C08929=1054.742,-26.097,429.977,170.873,29.984,155.636
C08930=1054.736,-26.347,429.991,170.872,29.982,155.635
C08931=1054.730,-26.597,430.005,170.871,29.980,155.635
C08932=1054.723,-26.846,430.018,170.869,29.978,155.635
C08933=1054.717,-27.095,430.031,170.867,29.976,155.635
C08934=1054.711,-27.345,430.045,170.865,29.974,155.634
C08935=1054.705,-27.595,430.059,170.864,29.972,155.634
C08936=1054.699,-27.844,430.072,170.862,29.971,155.634
C08937=1054.692,-28.094,430.086,170.860,29.968,155.634
C08938=1054.686,-28.343,430.099,170.858,29.967,155.634
C08939=1054.679,-28.592,430.112,170.856,29.965,155.633
C08940=1054.674,-28.842,430.125,170.855,29.963,155.633
C08941=1054.667,-29.092,430.138,170.853,29.961,155.633
C08942=1054.661,-29.342,430.152,170.851,29.959,155.633
C08943=1054.655,-29.591,430.165,170.849,29.958,155.633
C08944=1054.649,-29.840,430.179,170.847,29.956,155.632
C08945=1054.642,-30.090,430.192,170.846,29.954,155.632
C08946=1054.636,-30.340,430.206,170.844,29.952,155.632
C08947=1054.630,-30.589,430.218,170.843,29.950,155.632
C08948=1054.624,-30.839,430.231,170.841,29.949,155.632
C08949=1054.617,-31.089,430.245,170.839,29.947,155.631
C08950=1054.611,-31.338,430.258,170.838,29.945,155.631
C08951=1054.605,-31.587,430.272,170.836,29.943,155.631
C08952=1054.599,-31.837,430.285,170.834,29.941,155.631
C08953=1054.593,-32.087,430.298,170.832,29.940,155.631
C08954=1054.586,-32.337,430.312,170.830,29.938,155.630
C08955=1054.580,-32.586,430.325,170.829,29.936,155.630
C08956=1054.574,-32.836,430.338,170.827,29.934,155.630
C08957=1054.568,-33.085,430.351,170.825,29.932,155.630
C08958=1054.562,-33.334,430.364,170.823,29.931,155.630
C08959=1054.555,-33.584,430.378,170.821,29.928,155.629
C08960=1054.549,-33.834,430.390,170.820,29.927,155.629
C08961=1054.543,-34.083,430.404,170.818,29.925,155.629
C08962=1054.536,-34.363,430.418,170.816,29.923,155.629
C08963=1054.529,-34.643,430.433,170.814,29.921,155.628
C08964=1054.522,-34.922,430.448,170.812,29.919,155.628
C08965=1054.515,-35.202,430.463,170.810,29.917,155.628
C08966=1054.509,-35.452,430.476,170.808,29.915,155.628
C08967=1054.503,-35.702,430.489,170.806,29.913,155.628
C08968=1054.497,-35.951,430.503,170.805,29.912,155.627
C08969=1054.491,-36.201,430.515,170.803,29.910,155.627
C08970=1054.485,-36.450,430.529,170.802,29.908,155.627
C08971=1054.479,-36.699,430.542,170.800,29.906,155.627
C08972=1054.472,-36.950,430.555,170.798,29.904,155.627
C08973=1054.466,-37.199,430.568,170.796,29.903,155.626
C08974=1054.460,-37.449,430.581,170.794,29.901,155.626
C08975=1054.454,-37.699,430.594,170.793,29.899,155.626
C08976=1054.448,-37.948,430.607,170.791,29.897,155.626
C08977=1054.442,-38.198,430.620,170.789,29.895,155.626
C08978=1054.436,-38.447,430.633,170.787,29.894,155.625
C08979=1054.430,-38.697,430.645,170.785,29.892,155.625
C08980=1054.424,-38.946,430.659,170.784,29.890,155.625
C08981=1054.418,-39.196,430.671,170.782,29.888,155.625
C08982=1054.410,-39.446,430.684,170.780,29.887,155.625
C08983=1054.404,-39.695,430.697,170.778,29.885,155.624
C08984=1054.398,-39.945,430.710,170.776,29.884,155.624
C08985=1054.392,-40.195,430.723,170.775,29.881,155.624
C08986=1054.386,-40.444,430.736,170.773,29.880,155.624
C08987=1054.380,-40.694,430.749,170.771,29.878,155.624
C08988=1054.373,-40.943,430.761,170.769,29.877,155.624
C08989=1054.367,-41.193,430.774,170.767,29.875,155.623
C08990=1054.361,-41.442,430.787,170.765,29.873,155.623
C08991=1054.355,-41.692,430.800,170.764,29.871,155.623
C08992=1054.349,-41.941,430.813,170.762,29.870,155.623
C08993=1054.341,-42.191,430.825,170.760,29.868,155.623
C08994=1054.335,-42.441,430.838,170.758,29.867,155.622
C08995=1054.329,-42.690,430.851,170.756,29.864,155.622
C08996=1054.323,-42.940,430.864,170.755,29.863,155.622
C08997=1054.317,-43.190,430.877,170.753,29.861,155.622
C08998=1054.311,-43.439,430.889,170.751,29.860,155.622
C08999=1054.304,-43.688,430.902,170.749,29.858,155.622
C09000=1054.298,-43.938,430.915,170.747,29.856,155.621
C09001=1054.292,-44.188,430.928,170.746,29.854,155.621
C09002=1054.286,-44.437,430.940,170.744,29.853,155.621
C09003=1054.280,-44.687,430.952,170.742,29.851,155.621
C09004=1054.273,-44.936,430.966,170.740,29.849,155.621
C09005=1054.268,-45.186,430.978,170.738,29.848,155.621
C09006=1054.262,-45.436,430.991,170.736,29.846,155.620
C09007=1054.255,-45.685,431.004,170.735,29.845,155.620
C09008=1054.249,-45.935,431.016,170.733,29.843,155.620
C09009=1054.243,-46.185,431.029,170.731,29.841,155.620
C09010=1054.237,-46.434,431.042,170.729,29.839,155.620
C09011=1054.231,-46.684,431.054,170.727,29.838,155.619
C09012=1054.224,-46.933,431.066,170.726,29.836,155.619
C09013=1054.218,-47.183,431.079,170.724,29.835,155.619
C09014=1054.212,-47.433,431.092,170.722,29.833,155.619
C09015=1054.206,-47.683,431.105,170.720,29.831,155.619
C09016=1054.199,-47.932,431.117,170.718,29.829,155.619
C09017=1054.193,-48.181,431.130,170.717,29.828,155.618
C09018=1054.187,-48.431,431.142,170.715,29.826,155.618
C09019=1054.182,-48.680,431.155,170.713,29.825,155.618
C09020=1054.175,-48.930,431.167,170.711,29.823,155.618
C09021=1054.169,-49.180,431.179,170.709,29.821,155.618
C09022=1054.163,-49.429,431.192,170.707,29.820,155.618
C09023=1054.157,-49.679,431.205,170.706,29.818,155.618
C09024=1054.151,-49.929,431.217,170.704,29.817,155.617
C09025=1054.145,-50.178,431.230,170.702,29.815,155.617
C09026=1054.138,-50.459,431.244,170.700,29.813,155.617
C09027=1054.131,-50.738,431.257,170.697,29.811,155.617
C09028=1054.124,-51.019,431.271,170.696,29.809,155.617
C09029=1054.117,-51.299,431.285,170.694,29.808,155.616
C09030=1054.110,-51.549,431.297,170.692,29.806,155.616
C09031=1054.104,-51.798,431.310,170.690,29.805,155.616
C09032=1054.097,-52.048,431.322,170.688,29.803,155.616
C09033=1054.091,-52.298,431.335,170.687,29.802,155.616
C09034=1054.084,-52.547,431.347,170.685,29.801,155.616
C09035=1054.079,-52.797,431.359,170.683,29.799,155.616
C09036=1054.072,-53.047,431.371,170.681,29.797,155.616
C09037=1054.065,-53.296,431.383,170.679,29.796,155.615
C09038=1054.059,-53.546,431.396,170.677,29.794,155.615
C09039=1054.053,-53.795,431.407,170.676,29.793,155.615
C09040=1054.047,-54.045,431.420,170.673,29.791,155.615
C09041=1054.041,-54.294,431.432,170.671,29.790,155.615
C09042=1054.034,-54.544,431.444,170.669,29.788,155.615
C09043=1054.028,-54.794,431.456,170.667,29.787,155.615
C09044=1054.022,-55.043,431.468,170.666,29.785,155.614
C09045=1054.016,-55.293,431.481,170.664,29.784,155.614
C09046=1054.009,-55.543,431.493,170.662,29.783,155.614
C09047=1054.002,-55.793,431.505,170.660,29.781,155.614
C09048=1053.996,-56.042,431.517,170.658,29.779,155.614
C09049=1053.990,-56.291,431.529,170.656,29.778,155.614
C09050=1053.984,-56.541,431.541,170.655,29.776,155.614
C09051=1053.978,-56.791,431.553,170.653,29.775,155.614
C09052=1053.971,-57.040,431.565,170.651,29.774,155.613
C09053=1053.965,-57.290,431.578,170.649,29.772,155.613
C09054=1053.959,-57.540,431.590,170.647,29.770,155.613
C09055=1053.952,-57.789,431.602,170.645,29.769,155.613
C09056=1053.947,-58.038,431.614,170.644,29.768,155.613
C09057=1053.940,-58.288,431.626,170.642,29.766,155.613
C09058=1053.934,-58.538,431.638,170.640,29.765,155.613
C09059=1053.928,-58.788,431.650,170.638,29.763,155.612
C09060=1053.921,-59.038,431.662,170.636,29.761,155.612
C09061=1053.915,-59.288,431.674,170.634,29.760,155.612
C09062=1053.909,-59.536,431.686,170.632,29.759,155.612
C09063=1053.903,-59.786,431.698,170.630,29.757,155.612
C09064=1053.897,-60.036,431.710,170.628,29.756,155.612
C09065=1053.890,-60.285,431.722,170.626,29.755,155.612
C09066=1053.884,-60.535,431.733,170.624,29.753,155.612
C09067=1053.878,-60.785,431.746,170.623,29.751,155.611
C09068=1053.872,-61.034,431.758,170.621,29.750,155.611
C09069=1053.865,-61.284,431.770,170.619,29.749,155.611
C09070=1053.859,-61.534,431.782,170.617,29.747,155.611
C09071=1053.853,-61.783,431.793,170.615,29.746,155.611
C09072=1053.847,-62.033,431.805,170.613,29.745,155.611
C09073=1053.841,-62.283,431.818,170.612,29.743,155.611
C09074=1053.834,-62.532,431.830,170.610,29.741,155.611
C09075=1053.828,-62.781,431.841,170.608,29.740,155.610
C09076=1053.823,-63.032,431.853,170.606,29.739,155.610
C09077=1053.816,-63.281,431.865,170.604,29.737,155.610
C09078=1053.809,-63.531,431.877,170.601,29.736,155.610
C09079=1053.804,-63.780,431.889,170.600,29.735,155.610
C09080=1053.798,-64.030,431.900,170.598,29.733,155.610
C09081=1053.791,-64.280,431.912,170.596,29.731,155.610
C09082=1053.786,-64.529,431.924,170.594,29.730,155.610
C09083=1053.779,-64.779,431.936,170.592,29.729,155.610
C09084=1053.773,-65.029,431.948,170.591,29.727,155.609
C09085=1053.767,-65.278,431.959,170.589,29.726,155.609
C09086=1053.761,-65.528,431.971,170.587,29.725,155.609
C09087=1053.754,-65.778,431.983,170.585,29.723,155.609
C09088=1053.748,-66.027,431.995,170.583,29.721,155.609
C09089=1053.743,-66.277,432.007,170.581,29.720,155.609
C09090=1053.735,-66.559,432.020,170.579,29.719,155.609
C09091=1053.728,-66.840,432.033,170.577,29.717,155.609
C09092=1053.722,-67.122,432.046,170.575,29.715,155.608
C09093=1053.714,-67.403,432.059,170.572,29.714,155.608
C09094=1053.708,-67.652,432.071,170.570,29.713,155.608
C09095=1053.703,-67.903,432.083,170.568,29.711,155.608
C09096=1053.697,-68.152,432.094,170.567,29.709,155.608
C09097=1053.690,-68.401,432.106,170.565,29.709,155.608
C09098=1053.684,-68.652,432.118,170.563,29.707,155.608
C09099=1053.678,-68.900,432.130,170.561,29.705,155.608
C09100=1053.672,-69.151,432.141,170.559,29.704,155.608
C09101=1053.666,-69.400,432.153,170.557,29.703,155.607
C09102=1053.660,-69.650,432.165,170.556,29.702,155.607
C09103=1053.654,-69.900,432.176,170.554,29.700,155.607
C09104=1053.648,-70.149,432.187,170.552,29.699,155.607
C09105=1053.641,-70.399,432.199,170.549,29.697,155.607
C09106=1053.636,-70.648,432.211,170.547,29.696,155.607
C09107=1053.630,-70.898,432.223,170.545,29.695,155.607
